// TwinCAT 3 PLC project PLC1
// Title: Project Title
// Company: Company Name
// ProjectVersion: 0.0.1.1
// ProgramVersion: 3.1.4024.0
// CompilerDefines: VISU_USEWSTRING
// libraries:
//   CmpBitmapPool, * (System)
//   FloatingPointUtils, * (System)
//   Tc2_EtherCAT, * (Beckhoff Automation GmbH)
//   Tc2_Math, * (Beckhoff Automation GmbH)
//   Tc2_MC2, * (Beckhoff Automation GmbH)
//   Tc2_Standard, * (Beckhoff Automation GmbH)
//   Tc2_System, * (Beckhoff Automation GmbH)
//   Tc2_Utilities, * (Beckhoff Automation GmbH)
//   Tc3_Module, * (Beckhoff Automation GmbH)
//   VisuDialogs, * (System)
//   Util,3.5.11.0,System
//   VisuSymbols,3.5.10.0,System
// project tree:
//   Data Collection/dataAnalyse/ E_BoxResultCode.TcDUT, E_WallEntryRule.TcDUT, FB_Window.TcPOU, prgDataAnaylse.TcPOU, ST_BoxCorner.TcDUT, ST_WallPermission.TcDUT
//   Data Collection/ dataGrab.TcGVL, Dat_550_DataAxis.TcVIS, prgDataGrab.TcPOU, structAnalysis.TcDUT, typeDataAxis.TcDUT, typeVectorOptions.TcDUT
//   Data Collection/dynamicBox/ diaDataBox.TcVIS, FB_BoxControl.TcPOU, structBoxData.TcDUT, textListLeft.TcTLO, textListRight.TcTLO, textListTop.TcTLO, textListBottom.TcTLO
//   Data Collection/task/ DataGrab_1.TcTTO, taskDataGrab.TcPOU, typePoints.TcDUT
//   HMI1/Data/ gLicenceView.TcGVL, gModeAlternate.TcGVL, ManualPageTitle.TcTLO, ModeRowText.TcTLO, ScreenNames.TcTLO, stationLinked.TcTLO, TaskText.TcTLO, CycleType.TcTLO, FaultState.TcTLO, flag.TcIPO (not stored), FlasherCorner.TcIPO (not stored), gHMIButtons.TcGVL, gHMIDataConst.TcGVL, gHMIMotionRows.TcGVL, gHMIUnits.TcGVL, gMsgView.TcGVL, HMIColour.TcGVL, HomeState.TcTLO, ModeStates.TcTLO, ModeStatesHeader.TcTLO, UnitRowText.TcTLO, MotionRowText.TcTLO, LanguageRowText.TcTLO, gHMIData.TcGVL, MotionRowImages.TcIPO (not stored)
//   HMI1/Data/TOAST-HMI/ gTOASTHMI.TcGVL, structHMI.TcDUT, structHMIBtns.TcDUT, structHMIGlobal.TcDUT, structHMIMessages.TcDUT
//   HMI1/Logic/ FB_ReadTextList.TcPOU, prgHMIaxis.TcPOU, prgModeRows.TcPOU, prgMotionRow.TcPOU, VisuInit.TcPOU, FB_FindTextIndexNum.TcPOU, FB_FindTextLangText.TcPOU, FC_Setup.TcPOU, pouHMI.TcPOU, prgHMIcontrol.TcPOU, prgHMIstations.TcPOU, prgHMIUnits.TcPOU, prgHMILanguage.TcPOU, prgReadTextList.TcPOU, prgShowButtons.TcPOU
//   HMI1/Screens/Diagnostic Fieldbus/EtherCAT/ diagEtherCATSlave.TcVIS (not stored), diagEtherCATSlaveDetail.TcVIS (not stored), Dia_801_EtherCAT.TcVIS (not stored)
//   HMI1/Screens/Diagnostic Fieldbus/PROFIBUS/ diagDPhelp.TcVIS (not stored), diagDPSlave.TcVIS (not stored), Dia_802_Profibus.TcVIS (not stored)
//   HMI1/Screens/Diagnostic Fieldbus/PROFINET/ diagProfiNetSlaveDetail.TcVIS (not stored), diagProfiNetSlave.TcVIS (not stored), Dia_803_ProfiNet.TcVIS (not stored)
//   HMI1/Screens/Diagnostic IO View/ Dia_800_DataDisplay.TcVIS
//   HMI1/Screens/Dialogs/ dialogEnterValueInteger.TcVIS, dialogReject.TcVIS, dialogDeviceInfo.TcVIS, dialogGetLicensesEx.TcVIS, dialogEnterValue.TcVIS, visuDataDisplay.TcVIS, visuTaskData.TcVIS, dialogStation.TcVIS
//   HMI1/Screens/Layout/ Lay_040_MachineLayout.TcVIS
//   HMI1/Screens/Machine Settings/ constCSV.TcGVL, FB_ReadParams.TcPOU, FB_WriteParams.TcPOU, MachineSettings.TcGVL, MaS_800_SettingScreen.TcVIS, pouMachineSettings.TcPOU, typeRecord.TcDUT, typeSettings.TcDUT
//   HMI1/Screens/Menu/ Men_030_MenuScreen.TcVIS, Men_031_MenuScreen_2.TcVIS, Men_032_MenuScreen_3.TcVIS
//   HMI1/Screens/Messages/ Msg_020_Alarms.TcVIS, Msg_021_AlarmsView.TcVIS
//   HMI1/Screens/Mode/ Mod_001_ModeScreen.TcVIS, Mod_101_ModeScreen_Alternate.TcVIS, Mod_002_ModeScreenRows.TcVIS
//   HMI1/Screens/Motion/ Mot_010_Motions.TcVIS, Mot_011_Axis.TcVIS
//   HMI1/Screens/Popup/ PopupMenu1.TcVIS, PopupMenu2.TcVIS, PopupMenu3.TcVIS, PopupMenu4.TcVIS, PopupMenu5.TcVIS, popup_test.TcVIS (not stored)
//   HMI1/Screens/Process/ Prc_500_Part.TcVIS (not stored), Prc_501_Cycle.TcVIS (not stored)
//   HMI1/Screens/Safety/ Saf_700_SafetyStatus.TcVIS (not stored), Saf_701_SafetyChecksum.TcVIS (not stored), visuSafetyRow.TcVIS (not stored)
//   HMI1/Screens/Sequences/ AutoRowsVisu.TcGVL, SeqTest.TcVIS (not stored)
//   HMI1/Screens/System/ Sys_900_About.TcVIS (not stored), Sys_902_Version.TcVIS (not stored), Sys_901_HMISystem.TcVIS (not stored)
//   HMI1/Screens/Units/ Unt_401_Units.TcVIS (not stored), Unt_402_Axis.TcVIS (not stored), Unt_403_Language.TcVIS (not stored)
//   HMI1/Screens/Web/ Web_300_Browser.TcVIS (not stored)
//   HMI1/Templates/ AxisRow.TcVIS, LanguageRow.TcVIS, ModeRow.TcVIS, Tmp_001_Template_Alternate.TcVIS, UnitRow.TcVIS, MotionRow.TcVIS, Tmp_000_Template.TcVIS, MessageRow.TcVIS
//   PLC/FBs/Diagnostic/EtherCAT/ enumEtherCATstate.TcGVL (not stored), enumEtherCATSuffix.TcGVL (not stored), etherCATdiag.TcGVL (not stored), ethercatImages.TcIPO (not stored), etherCATmasters.TcGVL (not stored), FB_CheckEC_CRC_errors.TcPOU (not stored), FB_DecodeEtherCAT.TcPOU (not stored), pouEtherCATDiag.TcPOU (not stored)
//   PLC/FBs/Diagnostic/Profibus/ pouDPDiag.TcPOU (not stored), profibusDiag.TcGVL (not stored), profibusImages.TcIPO (not stored)
//   PLC/FBs/Diagnostic/ProfiNet/ enumProfiNetState.TcGVL (not stored), enumProfiNetSuffix.TcGVL (not stored), FB_DecodePROFINET.TcPOU (not stored), pouPROFINETdiag.TcPOU (not stored), ProfiNetDiag.TcGVL (not stored), ProfiNETImages.TcIPO (not stored)
//   PLC/FBs/FBs/ FB_ApplyLocks.TcPOU (not stored), FB_CheckAnyMode.TcPOU (not stored), FB_Flasher.TcPOU, FB_HMI_Control_NoGroupRef.TcPOU (not stored), FB_PowerDelay.TcPOU (not stored), FB_StationStats.TcPOU (not stored), FB_Step.TcPOU (not stored), FB_CheckMessageBounds.TcPOU (not stored), FB_HMI_Control.TcPOU (not stored), FB_Mode.TcPOU (not stored), FB_PartBuild.TcPOU (not stored), FB_ModeStateToColour.TcPOU (not stored)
//   PLC/FBs/FCs/ FC_NOT.TcPOU (not stored)
//   PLC/FBs/IO View/ FB_DataCombine.TcPOU (not stored), ioView.TcGVL (not stored), pouDataDisplay.TcPOU (not stored), prgMemPointerView.TcPOU (not stored)
//   PLC/FBs/Robot/ FB_RobotComms.TcPOU (not stored), FB_RobotMotion.TcPOU (not stored), robotCall.TcPOU (not stored), robotGlobals.TcGVL (not stored), structRobot.TcDUT (not stored), structRobotInputs.TcDUT (not stored), structRobotOutputs.TcDUT (not stored)
//   PLC/FBs/Sequence/ typeAutoRowMotion.TcDUT (not stored), AutoRows.TcGVL (not stored), FB_GetStateAutoRow.TcPOU (not stored), typeRowHolder.TcDUT (not stored), typeSeqRow.TcDUT (not stored)
//   PLC/FBs/Tasks/ FB_CheckTasks.TcPOU (not stored), FB_Task.TcPOU (not stored), FC_S1_AssignTaskTimes.TcPOU (not stored), FC_S2_AssignTaskTimes.TcPOU (not stored), FC_S3_AssignTaskTimes.TcPOU (not stored), FC_S4_AssignTaskTimes.TcPOU (not stored), FC_S5_AssignTaskTimes.TcPOU (not stored), FC_S6_AssignTaskTimes.TcPOU (not stored)
//   PLC/Machine/Base/ Mc_Variant.TcGVL (not stored), Mc_Global.TcGVL (not stored), pouMachine.TcPOU (not stored)
//   PLC/Machine/Station 1/Motions/Screen 10/ S1_01_Motion_89.TcPOU (not stored), S1_01_Motion_90.TcPOU (not stored), S1_01_Motion_91.TcPOU (not stored), S1_01_Motion_92.TcPOU (not stored), S1_01_Motion_93.TcPOU (not stored), S1_01_Motion_94.TcPOU (not stored), S1_01_Motion_95.TcPOU (not stored), S1_01_Motion_96.TcPOU (not stored), S1_01_Motion_97.TcPOU (not stored), S1_01_Motion_98.TcPOU (not stored), S1_01_Motion_99.TcPOU (not stored)
//   PLC/Machine/Station 1/Motions/Screen 1/ S1_01_RobPickPart_1.TcPOU (not stored), S1_01_RobClamp1_2.TcPOU (not stored), S1_01_RobClamp2_3.TcPOU (not stored), S1_01_RobWash_4.TcPOU (not stored), S1_01_WasherJets_5.TcPOU (not stored), S1_01_RobMarker_6.TcPOU (not stored), S1_01_MarkPart_7.TcPOU (not stored), S1_01_Motion_8.TcPOU (not stored), S1_01_Motion_9.TcPOU (not stored)
//   PLC/Machine/Station 1/Motions/Screen 2/ S1_01_Motion_10.TcPOU (not stored), S1_01_Motion_11.TcPOU (not stored), S1_01_Motion_12.TcPOU (not stored), S1_01_Motion_13.TcPOU (not stored), S1_01_Motion_14.TcPOU (not stored), S1_01_Motion_15.TcPOU (not stored), S1_01_Motion_16.TcPOU (not stored), S1_01_Motion_17.TcPOU (not stored), S1_01_Motion_18.TcPOU (not stored), S1_01_Motion_19.TcPOU (not stored)
//   PLC/Machine/Station 1/Motions/Screen 3/ S1_01_Motion_20.TcPOU (not stored), S1_01_Motion_21.TcPOU (not stored), S1_01_Motion_22.TcPOU (not stored), S1_01_Motion_23.TcPOU (not stored), S1_01_Motion_24.TcPOU (not stored), S1_01_Motion_25.TcPOU (not stored), S1_01_Motion_26.TcPOU (not stored), S1_01_Motion_27.TcPOU (not stored), S1_01_Motion_28.TcPOU (not stored)
//   PLC/Machine/Station 1/Motions/Screen 4/ S1_01_Motion_29.TcPOU (not stored), S1_01_Motion_30.TcPOU (not stored), S1_01_Motion_31.TcPOU (not stored), S1_01_Motion_32.TcPOU (not stored), S1_01_Motion_33.TcPOU (not stored), S1_01_Motion_34.TcPOU (not stored), S1_01_Motion_35.TcPOU (not stored), S1_01_Motion_36.TcPOU (not stored), S1_01_Motion_37.TcPOU (not stored), S1_01_Motion_38.TcPOU (not stored)
//   PLC/Machine/Station 1/Motions/Screen 5/ S1_01_Motion_39.TcPOU (not stored), S1_01_Motion_40.TcPOU (not stored), S1_01_Motion_41.TcPOU (not stored), S1_01_Motion_42.TcPOU (not stored), S1_01_Motion_43.TcPOU (not stored), S1_01_Motion_44.TcPOU (not stored), S1_01_Motion_45.TcPOU (not stored), S1_01_Motion_46.TcPOU (not stored), S1_01_Motion_47.TcPOU (not stored), S1_01_Motion_48.TcPOU (not stored)
//   PLC/Machine/Station 1/Motions/Screen 6/ S1_01_Motion_49.TcPOU (not stored), S1_01_Motion_50.TcPOU (not stored), S1_01_Motion_51.TcPOU (not stored), S1_01_Motion_52.TcPOU (not stored), S1_01_Motion_53.TcPOU (not stored), S1_01_Motion_54.TcPOU (not stored), S1_01_Motion_55.TcPOU (not stored), S1_01_Motion_56.TcPOU (not stored), S1_01_Motion_57.TcPOU (not stored), S1_01_Motion_58.TcPOU (not stored)
//   PLC/Machine/Station 1/Motions/Screen 7/ S1_01_Motion_59.TcPOU (not stored), S1_01_Motion_60.TcPOU (not stored), S1_01_Motion_61.TcPOU (not stored), S1_01_Motion_62.TcPOU (not stored), S1_01_Motion_63.TcPOU (not stored), S1_01_Motion_64.TcPOU (not stored), S1_01_Motion_65.TcPOU (not stored), S1_01_Motion_66.TcPOU (not stored), S1_01_Motion_67.TcPOU (not stored), S1_01_Motion_68.TcPOU (not stored)
//   PLC/Machine/Station 1/Motions/Screen 8/ S1_01_Motion_69.TcPOU (not stored), S1_01_Motion_70.TcPOU (not stored), S1_01_Motion_71.TcPOU (not stored), S1_01_Motion_72.TcPOU (not stored), S1_01_Motion_73.TcPOU (not stored), S1_01_Motion_74.TcPOU (not stored), S1_01_Motion_75.TcPOU (not stored), S1_01_Motion_76.TcPOU (not stored), S1_01_Motion_77.TcPOU (not stored), S1_01_Motion_78.TcPOU (not stored)
//   PLC/Machine/Station 1/Motions/Screen 9/ S1_01_Motion_79.TcPOU (not stored), S1_01_Motion_80.TcPOU (not stored), S1_01_Motion_81.TcPOU (not stored), S1_01_Motion_82.TcPOU (not stored), S1_01_Motion_83.TcPOU (not stored), S1_01_Motion_84.TcPOU (not stored), S1_01_Motion_85.TcPOU (not stored), S1_01_Motion_86.TcPOU (not stored), S1_01_Motion_87.TcPOU (not stored), S1_01_Motion_88.TcPOU (not stored)
//   PLC/Machine/Station 1/Sequence/ FB_S1_Sequence.TcPOU (not stored), S1sfc.TcGVL (not stored), struct_SFC_Row.TcDUT (not stored)
//   PLC/Machine/Station 2/Motions/Screen 10/ S2_01_Motion_89.TcPOU (not stored), S2_01_Motion_90.TcPOU (not stored), S2_01_Motion_91.TcPOU (not stored), S2_01_Motion_92.TcPOU (not stored), S2_01_Motion_93.TcPOU (not stored), S2_01_Motion_94.TcPOU (not stored), S2_01_Motion_95.TcPOU (not stored), S2_01_Motion_96.TcPOU (not stored), S2_01_Motion_97.TcPOU (not stored), S2_01_Motion_98.TcPOU (not stored), S2_01_Motion_99.TcPOU (not stored)
//   PLC/Machine/Station 2/Motions/Screen 1/ S2_01_Motion_1.TcPOU (not stored), S2_01_Motion_2.TcPOU (not stored), S2_01_Motion_3.TcPOU (not stored), S2_01_Motion_4.TcPOU (not stored), S2_01_Motion_5.TcPOU (not stored), S2_01_Motion_6.TcPOU (not stored), S2_01_Motion_7.TcPOU (not stored), S2_01_Motion_8.TcPOU (not stored), S2_01_Motion_9.TcPOU (not stored)
//   PLC/Machine/Station 2/Motions/Screen 2/ S2_01_Motion_10.TcPOU (not stored), S2_01_Motion_11.TcPOU (not stored), S2_01_Motion_12.TcPOU (not stored), S2_01_Motion_13.TcPOU (not stored), S2_01_Motion_14.TcPOU (not stored), S2_01_Motion_15.TcPOU (not stored), S2_01_Motion_16.TcPOU (not stored), S2_01_Motion_17.TcPOU (not stored), S2_01_Motion_18.TcPOU (not stored), S2_01_Motion_19.TcPOU (not stored)
//   PLC/Machine/Station 2/Motions/Screen 3/ S2_01_Motion_20.TcPOU (not stored), S2_01_Motion_21.TcPOU (not stored), S2_01_Motion_22.TcPOU (not stored), S2_01_Motion_23.TcPOU (not stored), S2_01_Motion_24.TcPOU (not stored), S2_01_Motion_25.TcPOU (not stored), S2_01_Motion_26.TcPOU (not stored), S2_01_Motion_27.TcPOU (not stored), S2_01_Motion_28.TcPOU (not stored)
//   PLC/Machine/Station 2/Motions/Screen 4/ S2_01_Motion_29.TcPOU (not stored), S2_01_Motion_30.TcPOU (not stored), S2_01_Motion_31.TcPOU (not stored), S2_01_Motion_32.TcPOU (not stored), S2_01_Motion_33.TcPOU (not stored), S2_01_Motion_34.TcPOU (not stored), S2_01_Motion_35.TcPOU (not stored), S2_01_Motion_36.TcPOU (not stored), S2_01_Motion_37.TcPOU (not stored), S2_01_Motion_38.TcPOU (not stored)
//   PLC/Machine/Station 2/Motions/Screen 5/ S2_01_Motion_39.TcPOU (not stored), S2_01_Motion_40.TcPOU (not stored), S2_01_Motion_41.TcPOU (not stored), S2_01_Motion_42.TcPOU (not stored), S2_01_Motion_43.TcPOU (not stored), S2_01_Motion_44.TcPOU (not stored), S2_01_Motion_45.TcPOU (not stored), S2_01_Motion_46.TcPOU (not stored), S2_01_Motion_47.TcPOU (not stored), S2_01_Motion_48.TcPOU (not stored)
//   PLC/Machine/Station 2/Motions/Screen 6/ S2_01_Motion_49.TcPOU (not stored), S2_01_Motion_50.TcPOU (not stored), S2_01_Motion_51.TcPOU (not stored), S2_01_Motion_52.TcPOU (not stored), S2_01_Motion_53.TcPOU (not stored), S2_01_Motion_54.TcPOU (not stored), S2_01_Motion_55.TcPOU (not stored), S2_01_Motion_56.TcPOU (not stored), S2_01_Motion_57.TcPOU (not stored), S2_01_Motion_58.TcPOU (not stored)
//   PLC/Machine/Station 2/Motions/Screen 7/ S2_01_Motion_59.TcPOU (not stored), S2_01_Motion_60.TcPOU (not stored), S2_01_Motion_61.TcPOU (not stored), S2_01_Motion_62.TcPOU (not stored), S2_01_Motion_63.TcPOU (not stored), S2_01_Motion_64.TcPOU (not stored), S2_01_Motion_65.TcPOU (not stored), S2_01_Motion_66.TcPOU (not stored), S2_01_Motion_67.TcPOU (not stored), S2_01_Motion_68.TcPOU (not stored)
//   PLC/Machine/Station 2/Motions/Screen 8/ S2_01_Motion_69.TcPOU (not stored), S2_01_Motion_70.TcPOU (not stored), S2_01_Motion_71.TcPOU (not stored), S2_01_Motion_72.TcPOU (not stored), S2_01_Motion_73.TcPOU (not stored), S2_01_Motion_74.TcPOU (not stored), S2_01_Motion_75.TcPOU (not stored), S2_01_Motion_76.TcPOU (not stored), S2_01_Motion_77.TcPOU (not stored), S2_01_Motion_78.TcPOU (not stored)
//   PLC/Machine/Station 2/Motions/Screen 9/ S2_01_Motion_79.TcPOU (not stored), S2_01_Motion_80.TcPOU (not stored), S2_01_Motion_81.TcPOU (not stored), S2_01_Motion_82.TcPOU (not stored), S2_01_Motion_83.TcPOU (not stored), S2_01_Motion_84.TcPOU (not stored), S2_01_Motion_85.TcPOU (not stored), S2_01_Motion_86.TcPOU (not stored), S2_01_Motion_87.TcPOU (not stored), S2_01_Motion_88.TcPOU (not stored)
//   PLC/Machine/Station 3/Motions/Screen 10/ S3_01_Motion_89.TcPOU (not stored), S3_01_Motion_90.TcPOU (not stored), S3_01_Motion_91.TcPOU (not stored), S3_01_Motion_92.TcPOU (not stored), S3_01_Motion_93.TcPOU (not stored), S3_01_Motion_94.TcPOU (not stored), S3_01_Motion_95.TcPOU (not stored), S3_01_Motion_96.TcPOU (not stored), S3_01_Motion_97.TcPOU (not stored), S3_01_Motion_98.TcPOU (not stored), S3_01_Motion_99.TcPOU (not stored)
//   PLC/Machine/Station 3/Motions/Screen 1/ S3_01_Motion_1.TcPOU (not stored), S3_01_Motion_2.TcPOU (not stored), S3_01_Motion_3.TcPOU (not stored), S3_01_Motion_4.TcPOU (not stored), S3_01_Motion_5.TcPOU (not stored), S3_01_Motion_6.TcPOU (not stored), S3_01_Motion_7.TcPOU (not stored), S3_01_Motion_8.TcPOU (not stored), S3_01_Motion_9.TcPOU (not stored)
//   PLC/Machine/Station 3/Motions/Screen 2/ S3_01_Motion_10.TcPOU (not stored), S3_01_Motion_11.TcPOU (not stored), S3_01_Motion_12.TcPOU (not stored), S3_01_Motion_13.TcPOU (not stored), S3_01_Motion_14.TcPOU (not stored), S3_01_Motion_15.TcPOU (not stored), S3_01_Motion_16.TcPOU (not stored), S3_01_Motion_17.TcPOU (not stored), S3_01_Motion_18.TcPOU (not stored), S3_01_Motion_19.TcPOU (not stored)
//   PLC/Machine/Station 3/Motions/Screen 3/ S3_01_Motion_20.TcPOU (not stored), S3_01_Motion_21.TcPOU (not stored), S3_01_Motion_22.TcPOU (not stored), S3_01_Motion_23.TcPOU (not stored), S3_01_Motion_24.TcPOU (not stored), S3_01_Motion_25.TcPOU (not stored), S3_01_Motion_26.TcPOU (not stored), S3_01_Motion_27.TcPOU (not stored), S3_01_Motion_28.TcPOU (not stored)
//   PLC/Machine/Station 3/Motions/Screen 4/ S3_01_Motion_29.TcPOU (not stored), S3_01_Motion_30.TcPOU (not stored), S3_01_Motion_31.TcPOU (not stored), S3_01_Motion_32.TcPOU (not stored), S3_01_Motion_33.TcPOU (not stored), S3_01_Motion_34.TcPOU (not stored), S3_01_Motion_35.TcPOU (not stored), S3_01_Motion_36.TcPOU (not stored), S3_01_Motion_37.TcPOU (not stored), S3_01_Motion_38.TcPOU (not stored)
//   PLC/Machine/Station 3/Motions/Screen 5/ S3_01_Motion_39.TcPOU (not stored), S3_01_Motion_40.TcPOU (not stored), S3_01_Motion_41.TcPOU (not stored), S3_01_Motion_42.TcPOU (not stored), S3_01_Motion_43.TcPOU (not stored), S3_01_Motion_44.TcPOU (not stored), S3_01_Motion_45.TcPOU (not stored), S3_01_Motion_46.TcPOU (not stored), S3_01_Motion_47.TcPOU (not stored), S3_01_Motion_48.TcPOU (not stored)
//   PLC/Machine/Station 3/Motions/Screen 6/ S3_01_Motion_49.TcPOU (not stored), S3_01_Motion_50.TcPOU (not stored), S3_01_Motion_51.TcPOU (not stored), S3_01_Motion_52.TcPOU (not stored), S3_01_Motion_53.TcPOU (not stored), S3_01_Motion_54.TcPOU (not stored), S3_01_Motion_55.TcPOU (not stored), S3_01_Motion_56.TcPOU (not stored), S3_01_Motion_57.TcPOU (not stored), S3_01_Motion_58.TcPOU (not stored)
//   PLC/Machine/Station 3/Motions/Screen 7/ S3_01_Motion_59.TcPOU (not stored), S3_01_Motion_60.TcPOU (not stored), S3_01_Motion_61.TcPOU (not stored), S3_01_Motion_62.TcPOU (not stored), S3_01_Motion_63.TcPOU (not stored), S3_01_Motion_64.TcPOU (not stored), S3_01_Motion_65.TcPOU (not stored), S3_01_Motion_66.TcPOU (not stored), S3_01_Motion_67.TcPOU (not stored), S3_01_Motion_68.TcPOU (not stored)
//   PLC/Machine/Station 3/Motions/Screen 8/ S3_01_Motion_69.TcPOU (not stored), S3_01_Motion_70.TcPOU (not stored), S3_01_Motion_71.TcPOU (not stored), S3_01_Motion_72.TcPOU (not stored), S3_01_Motion_73.TcPOU (not stored), S3_01_Motion_74.TcPOU (not stored), S3_01_Motion_75.TcPOU (not stored), S3_01_Motion_76.TcPOU (not stored), S3_01_Motion_77.TcPOU (not stored), S3_01_Motion_78.TcPOU (not stored)
//   PLC/Machine/Station 3/Motions/Screen 9/ S3_01_Motion_79.TcPOU (not stored), S3_01_Motion_80.TcPOU (not stored), S3_01_Motion_81.TcPOU (not stored), S3_01_Motion_82.TcPOU (not stored), S3_01_Motion_83.TcPOU (not stored), S3_01_Motion_84.TcPOU (not stored), S3_01_Motion_85.TcPOU (not stored), S3_01_Motion_86.TcPOU (not stored), S3_01_Motion_87.TcPOU (not stored), S3_01_Motion_88.TcPOU (not stored)
//   PLC/Machine/Station 4/Motions/Screen 10/ S4_01_Motion_89.TcPOU (not stored), S4_01_Motion_90.TcPOU (not stored), S4_01_Motion_91.TcPOU (not stored), S4_01_Motion_92.TcPOU (not stored), S4_01_Motion_93.TcPOU (not stored), S4_01_Motion_94.TcPOU (not stored), S4_01_Motion_95.TcPOU (not stored), S4_01_Motion_96.TcPOU (not stored), S4_01_Motion_97.TcPOU (not stored), S4_01_Motion_98.TcPOU (not stored), S4_01_Motion_99.TcPOU (not stored)
//   PLC/Machine/Station 4/Motions/Screen 1/ S4_01_Motion_1.TcPOU (not stored), S4_01_Motion_2.TcPOU (not stored), S4_01_Motion_3.TcPOU (not stored), S4_01_Motion_4.TcPOU (not stored), S4_01_Motion_5.TcPOU (not stored), S4_01_Motion_6.TcPOU (not stored), S4_01_Motion_7.TcPOU (not stored), S4_01_Motion_8.TcPOU (not stored), S4_01_Motion_9.TcPOU (not stored)
//   PLC/Machine/Station 4/Motions/Screen 2/ S4_01_Motion_10.TcPOU (not stored), S4_01_Motion_11.TcPOU (not stored), S4_01_Motion_12.TcPOU (not stored), S4_01_Motion_13.TcPOU (not stored), S4_01_Motion_14.TcPOU (not stored), S4_01_Motion_15.TcPOU (not stored), S4_01_Motion_16.TcPOU (not stored), S4_01_Motion_17.TcPOU (not stored), S4_01_Motion_18.TcPOU (not stored), S4_01_Motion_19.TcPOU (not stored)
//   PLC/Machine/Station 4/Motions/Screen 3/ S4_01_Motion_20.TcPOU (not stored), S4_01_Motion_21.TcPOU (not stored), S4_01_Motion_22.TcPOU (not stored), S4_01_Motion_23.TcPOU (not stored), S4_01_Motion_24.TcPOU (not stored), S4_01_Motion_25.TcPOU (not stored), S4_01_Motion_26.TcPOU (not stored), S4_01_Motion_27.TcPOU (not stored), S4_01_Motion_28.TcPOU (not stored)
//   PLC/Machine/Station 4/Motions/Screen 4/ S4_01_Motion_29.TcPOU (not stored), S4_01_Motion_30.TcPOU (not stored), S4_01_Motion_31.TcPOU (not stored), S4_01_Motion_32.TcPOU (not stored), S4_01_Motion_33.TcPOU (not stored), S4_01_Motion_34.TcPOU (not stored), S4_01_Motion_35.TcPOU (not stored), S4_01_Motion_36.TcPOU (not stored), S4_01_Motion_37.TcPOU (not stored), S4_01_Motion_38.TcPOU (not stored)
//   PLC/Machine/Station 4/Motions/Screen 5/ S4_01_Motion_39.TcPOU (not stored), S4_01_Motion_40.TcPOU (not stored), S4_01_Motion_41.TcPOU (not stored), S4_01_Motion_42.TcPOU (not stored), S4_01_Motion_43.TcPOU (not stored), S4_01_Motion_44.TcPOU (not stored), S4_01_Motion_45.TcPOU (not stored), S4_01_Motion_46.TcPOU (not stored), S4_01_Motion_47.TcPOU (not stored), S4_01_Motion_48.TcPOU (not stored)
//   PLC/Machine/Station 4/Motions/Screen 6/ S4_01_Motion_49.TcPOU (not stored), S4_01_Motion_50.TcPOU (not stored), S4_01_Motion_51.TcPOU (not stored), S4_01_Motion_52.TcPOU (not stored), S4_01_Motion_53.TcPOU (not stored), S4_01_Motion_54.TcPOU (not stored), S4_01_Motion_55.TcPOU (not stored), S4_01_Motion_56.TcPOU (not stored), S4_01_Motion_57.TcPOU (not stored), S4_01_Motion_58.TcPOU (not stored)
//   PLC/Machine/Station 4/Motions/Screen 7/ S4_01_Motion_59.TcPOU (not stored), S4_01_Motion_60.TcPOU (not stored), S4_01_Motion_61.TcPOU (not stored), S4_01_Motion_62.TcPOU (not stored), S4_01_Motion_63.TcPOU (not stored), S4_01_Motion_64.TcPOU (not stored), S4_01_Motion_65.TcPOU (not stored), S4_01_Motion_66.TcPOU (not stored), S4_01_Motion_67.TcPOU (not stored), S4_01_Motion_68.TcPOU (not stored)
//   PLC/Machine/Station 4/Motions/Screen 8/ S4_01_Motion_69.TcPOU (not stored), S4_01_Motion_70.TcPOU (not stored), S4_01_Motion_71.TcPOU (not stored), S4_01_Motion_72.TcPOU (not stored), S4_01_Motion_73.TcPOU (not stored), S4_01_Motion_74.TcPOU (not stored), S4_01_Motion_75.TcPOU (not stored), S4_01_Motion_76.TcPOU (not stored), S4_01_Motion_77.TcPOU (not stored), S4_01_Motion_78.TcPOU (not stored)
//   PLC/Machine/Station 4/Motions/Screen 9/ S4_01_Motion_79.TcPOU (not stored), S4_01_Motion_80.TcPOU (not stored), S4_01_Motion_81.TcPOU (not stored), S4_01_Motion_82.TcPOU (not stored), S4_01_Motion_83.TcPOU (not stored), S4_01_Motion_84.TcPOU (not stored), S4_01_Motion_85.TcPOU (not stored), S4_01_Motion_86.TcPOU (not stored), S4_01_Motion_87.TcPOU (not stored), S4_01_Motion_88.TcPOU (not stored)
//   PLC/Machine/Station 5/Motions/Screen 10/ S5_01_Motion_89.TcPOU (not stored), S5_01_Motion_90.TcPOU (not stored), S5_01_Motion_91.TcPOU (not stored), S5_01_Motion_92.TcPOU (not stored), S5_01_Motion_93.TcPOU (not stored), S5_01_Motion_94.TcPOU (not stored), S5_01_Motion_95.TcPOU (not stored), S5_01_Motion_96.TcPOU (not stored), S5_01_Motion_97.TcPOU (not stored), S5_01_Motion_98.TcPOU (not stored), S5_01_Motion_99.TcPOU (not stored)
//   PLC/Machine/Station 5/Motions/Screen 1/ S5_01_Motion_1.TcPOU (not stored), S5_01_Motion_2.TcPOU (not stored), S5_01_Motion_3.TcPOU (not stored), S5_01_Motion_4.TcPOU (not stored), S5_01_Motion_5.TcPOU (not stored), S5_01_Motion_6.TcPOU (not stored), S5_01_Motion_7.TcPOU (not stored), S5_01_Motion_8.TcPOU (not stored), S5_01_Motion_9.TcPOU (not stored)
//   PLC/Machine/Station 5/Motions/Screen 2/ S5_01_Motion_10.TcPOU (not stored), S5_01_Motion_11.TcPOU (not stored), S5_01_Motion_12.TcPOU (not stored), S5_01_Motion_13.TcPOU (not stored), S5_01_Motion_14.TcPOU (not stored), S5_01_Motion_15.TcPOU (not stored), S5_01_Motion_16.TcPOU (not stored), S5_01_Motion_17.TcPOU (not stored), S5_01_Motion_18.TcPOU (not stored), S5_01_Motion_19.TcPOU (not stored)
//   PLC/Machine/Station 5/Motions/Screen 3/ S5_01_Motion_20.TcPOU (not stored), S5_01_Motion_21.TcPOU (not stored), S5_01_Motion_22.TcPOU (not stored), S5_01_Motion_23.TcPOU (not stored), S5_01_Motion_24.TcPOU (not stored), S5_01_Motion_25.TcPOU (not stored), S5_01_Motion_26.TcPOU (not stored), S5_01_Motion_27.TcPOU (not stored), S5_01_Motion_28.TcPOU (not stored), S5_01_Motion_29.TcPOU (not stored)
//   PLC/Machine/Station 5/Motions/Screen 4/ S5_01_Motion_30.TcPOU (not stored), S5_01_Motion_31.TcPOU (not stored), S5_01_Motion_32.TcPOU (not stored), S5_01_Motion_33.TcPOU (not stored), S5_01_Motion_34.TcPOU (not stored), S5_01_Motion_35.TcPOU (not stored), S5_01_Motion_36.TcPOU (not stored), S5_01_Motion_37.TcPOU (not stored), S5_01_Motion_38.TcPOU (not stored), S5_01_Motion_39.TcPOU (not stored)
//   PLC/Machine/Station 5/Motions/Screen 5/ S5_01_Motion_40.TcPOU (not stored), S5_01_Motion_41.TcPOU (not stored), S5_01_Motion_42.TcPOU (not stored), S5_01_Motion_43.TcPOU (not stored), S5_01_Motion_44.TcPOU (not stored), S5_01_Motion_45.TcPOU (not stored), S5_01_Motion_46.TcPOU (not stored), S5_01_Motion_47.TcPOU (not stored), S5_01_Motion_48.TcPOU (not stored), S5_01_Motion_49.TcPOU (not stored)
//   PLC/Machine/Station 5/Motions/Screen 6/ S5_01_Motion_50.TcPOU (not stored), S5_01_Motion_51.TcPOU (not stored), S5_01_Motion_52.TcPOU (not stored), S5_01_Motion_53.TcPOU (not stored), S5_01_Motion_54.TcPOU (not stored), S5_01_Motion_55.TcPOU (not stored), S5_01_Motion_56.TcPOU (not stored), S5_01_Motion_57.TcPOU (not stored), S5_01_Motion_58.TcPOU (not stored), S5_01_Motion_59.TcPOU (not stored)
//   PLC/Machine/Station 5/Motions/Screen 7/ S5_01_Motion_60.TcPOU (not stored), S5_01_Motion_61.TcPOU (not stored), S5_01_Motion_62.TcPOU (not stored), S5_01_Motion_63.TcPOU (not stored), S5_01_Motion_64.TcPOU (not stored), S5_01_Motion_65.TcPOU (not stored), S5_01_Motion_66.TcPOU (not stored), S5_01_Motion_67.TcPOU (not stored), S5_01_Motion_68.TcPOU (not stored), S5_01_Motion_69.TcPOU (not stored)
//   PLC/Machine/Station 5/Motions/Screen 8/ S5_01_Motion_70.TcPOU (not stored), S5_01_Motion_71.TcPOU (not stored), S5_01_Motion_72.TcPOU (not stored), S5_01_Motion_73.TcPOU (not stored), S5_01_Motion_74.TcPOU (not stored), S5_01_Motion_75.TcPOU (not stored), S5_01_Motion_76.TcPOU (not stored), S5_01_Motion_77.TcPOU (not stored), S5_01_Motion_78.TcPOU (not stored), S5_01_Motion_79.TcPOU (not stored)
//   PLC/Machine/Station 5/Motions/Screen 9/ S5_01_Motion_80.TcPOU (not stored), S5_01_Motion_81.TcPOU (not stored), S5_01_Motion_82.TcPOU (not stored), S5_01_Motion_83.TcPOU (not stored), S5_01_Motion_84.TcPOU (not stored), S5_01_Motion_85.TcPOU (not stored), S5_01_Motion_86.TcPOU (not stored), S5_01_Motion_87.TcPOU (not stored), S5_01_Motion_88.TcPOU (not stored)
//   PLC/Machine/Station 6/Motions/Screen 10/ S6_01_Motion_89.TcPOU (not stored), S6_01_Motion_90.TcPOU (not stored), S6_01_Motion_91.TcPOU (not stored), S6_01_Motion_92.TcPOU (not stored), S6_01_Motion_93.TcPOU (not stored), S6_01_Motion_94.TcPOU (not stored), S6_01_Motion_95.TcPOU (not stored), S6_01_Motion_96.TcPOU (not stored), S6_01_Motion_97.TcPOU (not stored), S6_01_Motion_98.TcPOU (not stored), S6_01_Motion_99.TcPOU (not stored)
//   PLC/Machine/Station 6/Motions/Screen 1/ S6_01_Motion_1.TcPOU (not stored), S6_01_Motion_2.TcPOU (not stored), S6_01_Motion_3.TcPOU (not stored), S6_01_Motion_4.TcPOU (not stored), S6_01_Motion_5.TcPOU (not stored), S6_01_Motion_6.TcPOU (not stored), S6_01_Motion_7.TcPOU (not stored), S6_01_Motion_8.TcPOU (not stored), S6_01_Motion_9.TcPOU (not stored)
//   PLC/Machine/Station 6/Motions/Screen 2/ S6_01_Motion_10.TcPOU (not stored), S6_01_Motion_11.TcPOU (not stored), S6_01_Motion_12.TcPOU (not stored), S6_01_Motion_13.TcPOU (not stored), S6_01_Motion_14.TcPOU (not stored), S6_01_Motion_15.TcPOU (not stored), S6_01_Motion_16.TcPOU (not stored), S6_01_Motion_17.TcPOU (not stored), S6_01_Motion_18.TcPOU (not stored), S6_01_Motion_19.TcPOU (not stored)
//   PLC/Machine/Station 6/Motions/Screen 3/ S6_01_Motion_20.TcPOU (not stored), S6_01_Motion_21.TcPOU (not stored), S6_01_Motion_22.TcPOU (not stored), S6_01_Motion_23.TcPOU (not stored), S6_01_Motion_24.TcPOU (not stored), S6_01_Motion_25.TcPOU (not stored), S6_01_Motion_26.TcPOU (not stored), S6_01_Motion_27.TcPOU (not stored), S6_01_Motion_28.TcPOU (not stored), S6_01_Motion_29.TcPOU (not stored)
//   PLC/Machine/Station 6/Motions/Screen 4/ S6_01_Motion_30.TcPOU (not stored), S6_01_Motion_31.TcPOU (not stored), S6_01_Motion_32.TcPOU (not stored), S6_01_Motion_33.TcPOU (not stored), S6_01_Motion_34.TcPOU (not stored), S6_01_Motion_35.TcPOU (not stored), S6_01_Motion_36.TcPOU (not stored), S6_01_Motion_37.TcPOU (not stored), S6_01_Motion_38.TcPOU (not stored), S6_01_Motion_39.TcPOU (not stored)
//   PLC/Machine/Station 6/Motions/Screen 5/ S6_01_Motion_40.TcPOU (not stored), S6_01_Motion_41.TcPOU (not stored), S6_01_Motion_42.TcPOU (not stored), S6_01_Motion_43.TcPOU (not stored), S6_01_Motion_44.TcPOU (not stored), S6_01_Motion_45.TcPOU (not stored), S6_01_Motion_46.TcPOU (not stored), S6_01_Motion_47.TcPOU (not stored), S6_01_Motion_48.TcPOU (not stored), S6_01_Motion_49.TcPOU (not stored)
//   PLC/Machine/Station 6/Motions/Screen 6/ S6_01_Motion_50.TcPOU (not stored), S6_01_Motion_51.TcPOU (not stored), S6_01_Motion_52.TcPOU (not stored), S6_01_Motion_53.TcPOU (not stored), S6_01_Motion_54.TcPOU (not stored), S6_01_Motion_55.TcPOU (not stored), S6_01_Motion_56.TcPOU (not stored), S6_01_Motion_57.TcPOU (not stored), S6_01_Motion_58.TcPOU (not stored), S6_01_Motion_59.TcPOU (not stored)
//   PLC/Machine/Station 6/Motions/Screen 7/ S6_01_Motion_60.TcPOU (not stored), S6_01_Motion_61.TcPOU (not stored), S6_01_Motion_62.TcPOU (not stored), S6_01_Motion_63.TcPOU (not stored), S6_01_Motion_64.TcPOU (not stored), S6_01_Motion_65.TcPOU (not stored), S6_01_Motion_66.TcPOU (not stored), S6_01_Motion_67.TcPOU (not stored), S6_01_Motion_68.TcPOU (not stored), S6_01_Motion_69.TcPOU (not stored)
//   PLC/Machine/Station 6/Motions/Screen 8/ S6_01_Motion_70.TcPOU (not stored), S6_01_Motion_71.TcPOU (not stored), S6_01_Motion_72.TcPOU (not stored), S6_01_Motion_73.TcPOU (not stored), S6_01_Motion_74.TcPOU (not stored), S6_01_Motion_75.TcPOU (not stored), S6_01_Motion_76.TcPOU (not stored), S6_01_Motion_77.TcPOU (not stored), S6_01_Motion_78.TcPOU (not stored), S6_01_Motion_79.TcPOU (not stored)
//   PLC/Machine/Station 6/Motions/Screen 9/ S6_01_Motion_80.TcPOU (not stored), S6_01_Motion_81.TcPOU (not stored), S6_01_Motion_82.TcPOU (not stored), S6_01_Motion_83.TcPOU (not stored), S6_01_Motion_84.TcPOU (not stored), S6_01_Motion_85.TcPOU (not stored), S6_01_Motion_86.TcPOU (not stored), S6_01_Motion_87.TcPOU (not stored), S6_01_Motion_88.TcPOU (not stored)
//   PLC/Safety/ enumEstopState.TcDUT, prgSafetyMain.TcPOU, Safety.TcGVL, structEstopDiag.TcDUT, structSafetyEstopDiagBOOList.TcDUT
//   PLC/System/ImplicitChecks/ CheckBounds.TcPOU (not stored), CheckDivDInt.TcPOU (not stored), CheckDivLInt.TcPOU (not stored), CheckDivLReal.TcPOU (not stored), CheckDivReal.TcPOU (not stored), CheckLRangeSigned.TcPOU (not stored), CheckLRangeUnsigned.TcPOU (not stored), CheckPointer.TcPOU (not stored), CheckRangeSigned.TcPOU (not stored), CheckRangeUnsigned.TcPOU (not stored)
//   Project Information/ F_GetCompany.TcPOU, F_GetTitle.TcPOU, F_GetVersion.TcPOU
//   Version/ Global_Version.TcGVL
//   X_DUTs/Diagnostic/ typeDPSlaveIndicator.TcDUT, typeEtherCATIndicator.TcDUT, typeEtherCATmasters.TcDUT, typeEtherCATState.TcDUT, typePROFINETIndicator.TcDUT, typeProfiNetMaster.TcDUT, typePROFINETState.TcDUT
//   X_DUTs/Drives/ HMIaxisDefinition.TcDUT, typeDriveInterface.TcDUT
//   X_DUTs/HMI/ typeBtnFdbk.TcDUT, typeBtnHides.TcDUT, typeBtnPress.TcDUT, typeHMIheader.TcDUT, typeMessageRow.TcDUT (not stored), typeMessageRowsArry.TcDUT, typeStationEnables.TcDUT (not stored)
//   X_DUTs/IO View/ dutDWord.TcDUT (not stored), typeCombineString.TcDUT (not stored)
//   X_DUTs/Langauge/ LanguageLocation.TcDUT (not stored)
//   X_DUTs/MessageView/ typeNewMsg.TcDUT, typeNewMsgHeader.TcDUT (not stored), typeNewMsgStyle.TcDUT
//   X_DUTs/Message/ typeAlarmViewStation.TcDUT (not stored), typeMessage.TcDUT (not stored), typeStationMessage.TcDUT (not stored), typeStationStatus.TcDUT (not stored)
//   X_DUTs/Motion/ RowConfig.TcDUT (not stored), typeMotionRecordRow.TcDUT, typeMotionRow.TcDUT, typeMotionRowArry.TcDUT, typeMotionRowButtons.TcDUT, typeMotionRowIO.TcDUT, typeMotionSide.TcDUT
//   X_DUTs/Screen/ typeMotionScreen.TcDUT, typeMotionScreenBtn.TcDUT
//   X_DUTs/Setup/ typeSetupMachine.TcDUT (not stored), typeSetupStation.TcDUT
//   X_DUTs/Station/ enumStationState.TcDUT, typeIndividualTask.TcDUT, typeRemote.TcDUT (not stored), typeStation.TcDUT, typeStationComplexity.TcDUT, typeStationComplexityBuffer.TcDUT, typeStationLockModes.TcDUT, typeStationLocks.TcDUT, typeStationMode.TcDUT, typeStationTask.TcDUT
//   / GlobalTextList.TcGTLO, PlcTask.TcTTO, Visualization Manager.TcVMO (not stored)
//   PLC/FBs/Drives/ driveGlobals.TcGVL (not stored), driveTestCall.TcPOU (not stored), FB_DriveInterface.TcPOU (not stored), FB_DriveMotion.TcPOU (not stored)
//   PLC/FBs/FBs/Motions/ FB_Motion1way.TcPOU (not stored), FB_Motion2way.TcPOU (not stored)
//   PLC/Machine/Base/Axis/ Axis.TcGVL (not stored), AxisRowText.TcTLO (not stored), pouAxis.TcPOU (not stored)
//   PLC/Machine/Base/Axis/RowAxis/ Ax_01_AxisIncrementSelect_04.TcPOU (not stored), Ax_01_AxisMoveAbsRel_06.TcPOU (not stored), Ax_01_AxisMoveJog_05.TcPOU (not stored), Ax_01_AxisMoveTypeSelect_02.TcPOU (not stored), Ax_01_AxisNameSelect_01.TcPOU (not stored), Ax_01_AxisSpeedSelect_03.TcPOU (not stored)
//   PLC/Machine/Base/Messages/Alarms/ pouMcAlarms.TcPOU (not stored)
//   PLC/Machine/Base/Messages/ pouMsgMc.TcPOU (not stored)
//   PLC/Machine/Base/Messages/Prompts/ pouMcPrompts.TcPOU (not stored)
//   PLC/Machine/Base/Messages/Warnings/ pouMcWarnings.TcPOU (not stored)
//   PLC/Machine/Base/Station Status/ AnyStationAlarmList.TcTLO (not stored), AnyStationWarningList.TcTLO (not stored), prgAfterStationScan.TcPOU (not stored), StationNames.TcTLO (not stored)
//   PLC/Machine/Base/Units/ Mc_01_Units_02.TcPOU (not stored), Mc_01_Units_03.TcPOU (not stored), Mc_01_Units_04.TcPOU (not stored), Mc_01_Units_05.TcPOU (not stored), Mc_01_Units_06.TcPOU (not stored), pouStationUnits.TcPOU (not stored), Mc_01_Units_01.TcPOU (not stored)
//   PLC/Machine/Base/Language/ Mc_02_Language_01.TcPOU (not stored), Mc_02_Language_02.TcPOU (not stored), Mc_02_Language_03.TcPOU (not stored), Mc_02_Language_04.TcPOU (not stored), Mc_02_Language_05.TcPOU (not stored), Mc_02_Language_06.TcPOU (not stored), pouStationLangauge.TcPOU (not stored)
//   PLC/Machine/ GlobalMessages.TcGVL, Remote.TcGVL, System.TcGVL
//   PLC/Machine/Station 2/Messages/Alarms/ pouS2Alarms.TcPOU (not stored)
//   PLC/Machine/Station 2/Messages/ pouMsgS2.TcPOU (not stored)
//   PLC/Machine/Station 2/Messages/Prompts/ pouS2Prompts.TcPOU (not stored)
//   PLC/Machine/Station 2/Messages/Warnings/ pouS2Warnings.TcPOU (not stored)
//   PLC/Machine/Station 2/ pouStation2.TcPOU (not stored), S2_Global.TcGVL (not stored), S2_IO.TcGVL (not stored)
//   PLC/Machine/Station 3/Messages/Alarms/ pouS3Alarms.TcPOU (not stored)
//   PLC/Machine/Station 3/Messages/ pouMsgS3.TcPOU (not stored)
//   PLC/Machine/Station 3/Messages/Prompts/ pouS3Prompts.TcPOU (not stored)
//   PLC/Machine/Station 3/Messages/Warnings/ pouS3Warnings.TcPOU (not stored)
//   PLC/Machine/Station 3/ pouStation3.TcPOU (not stored), S3_Global.TcGVL (not stored), S3_IO.TcGVL (not stored)
//   PLC/Machine/Station 4/Messages/Alarms/ pouS4Alarms.TcPOU (not stored)
//   PLC/Machine/Station 4/Messages/ pouMsgS4.TcPOU (not stored)
//   PLC/Machine/Station 4/Messages/Prompts/ pouS4Prompts.TcPOU (not stored)
//   PLC/Machine/Station 4/Messages/Warnings/ pouS4Warnings.TcPOU (not stored)
//   PLC/Machine/Station 4/ pouStation4.TcPOU (not stored), S4_Global.TcGVL (not stored), S4_IO.TcGVL (not stored)
//   PLC/Machine/Station 5/Messages/Alarms/ pouS5Alarms.TcPOU (not stored)
//   PLC/Machine/Station 5/Messages/ pouMsgS5.TcPOU (not stored)
//   PLC/Machine/Station 5/Messages/Prompts/ pouS5Prompts.TcPOU (not stored)
//   PLC/Machine/Station 5/Messages/Warnings/ pouS5Warnings.TcPOU (not stored)
//   PLC/Machine/Station 5/ pouStation5.TcPOU (not stored), S5_Global.TcGVL (not stored), S5_IO.TcGVL (not stored)
//   PLC/Machine/Station 6/Messages/Alarms/ pouS6Alarms.TcPOU (not stored)
//   PLC/Machine/Station 6/Messages/ pouMsgS6.TcPOU (not stored)
//   PLC/Machine/Station 6/Messages/Prompts/ pouS6Prompts.TcPOU (not stored)
//   PLC/Machine/Station 6/Messages/Warnings/ pouS6Warnings.TcPOU (not stored)
//   PLC/Machine/Station 6/ pouStation6.TcPOU (not stored), S6_Global.TcGVL (not stored), S6_IO.TcGVL (not stored)
//   PLC/Machine/Station 1/ S1_IO.TcGVL (not stored), pouStation1.TcPOU (not stored), S1_Global.TcGVL (not stored)
//   PLC/Machine/Station 1/Messages/Alarms/ pouS1Alarms.TcPOU (not stored)
//   PLC/Machine/Station 1/Messages/ pouMsgS1.TcPOU (not stored)
//   PLC/Machine/Station 1/Messages/Prompts/ pouS1Prompts.TcPOU (not stored)
//   PLC/Machine/Station 1/Messages/Warnings/ pouS1Warnings.TcPOU (not stored)
//   PLC/ MAIN.TcPOU
//   X_DUTs/Tasks/ Tasks.TcGVL, TaskState.TcDUT
//   X_Language Text/Messages/Machine/ Mc_Alarms.TcTLO (not stored), Mc_Prompts.TcTLO (not stored), Mc_Warnings.TcTLO (not stored)
//   X_Language Text/Messages/Station 1/ S1_Alarms.TcTLO (not stored), S1_Prompts.TcTLO (not stored), S1_Warnings.TcTLO (not stored)
//   X_Language Text/Messages/Station 2/ S2_Alarms.TcTLO (not stored), S2_Prompts.TcTLO (not stored), S2_Warnings.TcTLO (not stored)
//   X_Language Text/Messages/Station 3/ S3_Alarms.TcTLO (not stored), S3_Prompts.TcTLO (not stored), S3_Warnings.TcTLO (not stored)
//   X_Language Text/Messages/Station 4/ S4_Alarms.TcTLO (not stored), S4_Prompts.TcTLO (not stored), S4_Warnings.TcTLO (not stored)
//   X_Language Text/Messages/Station 5/ S5_Alarms.TcTLO (not stored), S5_Prompts.TcTLO (not stored), S5_Warnings.TcTLO (not stored)
//   X_Language Text/Messages/Station 6/ S6_Alarms.TcTLO (not stored), S6_Prompts.TcTLO (not stored), S6_Warnings.TcTLO (not stored)
//   X_Sim/ FB_SimMotion.TcPOU

CONFIGURATION PLC1
    RESOURCE PLC ON TwinCAT3
        TASK DataGrab_1(INTERVAL := T#1ms, PRIORITY := 4);
        TASK PlcTask(INTERVAL := T#10ms, PRIORITY := 14);
        PROGRAM taskDataGrab WITH DataGrab_1 : taskDataGrab;
        PROGRAM MAIN WITH PlcTask : MAIN;
    END_RESOURCE
END_CONFIGURATION

// ---- Data Collection/dataAnalyse/E_BoxResultCode.TcDUT
{attribute 'qualified_only'}
{attribute 'strict'}
TYPE E_BoxResultCode :
(
    Success                     := 0,  // Signal perfectly trapped inside the box
    Err_NeverEnteredBox         := 10, // Dataset finished, signal never entered the box boundaries
    Err_IllegalEntry_SideA      := 11, // Crossed Side A (Left) but it was configured as illegal
    Err_IllegalEntry_SideC      := 13, // Crossed Side C (Top) but it was configured as illegal
    Err_IllegalEntry_SideD      := 14, // Crossed Side D (Bottom) but it was configured as illegal
	Err_WrongEntryWall			:= 15, // Entered the wrong wall!
    
    Leak_Exited_SideA           := 21, // Signal backed out of Side A (Left Wall)
    Leak_Exited_SideB           := 22, // Signal broke out of Side B (Right Wall)
    Leak_Exited_SideC           := 23, // Signal spiked over the roof out of Side C (Top Wall)
    Leak_Exited_SideD           := 24, // Signal dropped out of the floor through Side D (Bottom Wall)
    
    Violation_Exited_SideA     := 31, // Signal left Side A which was explicitly locked via IsNotPermittedToExit
    Violation_Exited_SideB     := 32, // Signal left Side B which was explicitly locked via IsNotPermittedToExit
    Violation_Exited_SideC     := 33, // Signal left Side C which was explicitly locked via IsNotPermittedToExit
    Violation_Exited_SideD     := 34  // Signal left Side D which was explicitly locked via IsNotPermittedToExit

) INT;
END_TYPE

// ---- Data Collection/dataAnalyse/E_WallEntryRule.TcDUT
// ENUM to define entry wall strictness
TYPE E_WallEntryRule :
(
    NoCheck      := 0, // Anyone can enter here. Doesn't force or block data.
    MustEnter    := 1, // Trajectory MUST enter here. If it enters somewhere else first, it fails.
    MustNotEnter := 2  // Strict wall blocker. If trajectory touches this wall, it fails immediately.
) BYTE;
END_TYPE

// ---- Data Collection/dataAnalyse/ST_BoxCorner.TcDUT
TYPE ST_BoxCorner : 
	STRUCT 
		PointXTime : LREAL; 
		PointYValue : LREAL; 
	END_STRUCT
END_TYPE

// ---- Data Collection/dataAnalyse/ST_WallPermission.TcDUT
// The updated wall permission structure
TYPE ST_WallPermission :
STRUCT
    EntryRule            : E_WallEntryRule; // Rule type: NoCheck, MustEnter, or MustNotEnter
    IsNotPermittedToExit  : BOOL;           // TRUE if not permitted to exit
END_STRUCT
END_TYPE

// ---- Data Collection/dynamicBox/structBoxData.TcDUT
TYPE structBoxData :
STRUCT
	topStatus:ST_WallPermission;
	bottomStatus:ST_WallPermission;
	leftStatus:ST_WallPermission;
	rightStatus:ST_WallPermission;
	
	topStatusChange:BOOL;
	bottomStatusChange:BOOL;
	leftStatusChange:BOOL;
	rightStatusChange:BOOL;
	
	
	    // Corner Points
    i1 : ST_BoxCorner; // Top-Left
    i2 : ST_BoxCorner; // Bottom-Left
    i3 : ST_BoxCorner; // Bottom-Right
    i4 : ST_BoxCorner; // Top-Right
	
END_STRUCT
END_TYPE

// ---- Data Collection/structAnalysis.TcDUT
TYPE structAnalysis :
STRUCT
	axis:typeDataAxis; //the data itself
	box1:structBoxData;
	box2:structBoxData;
	box3:structBoxData;
END_STRUCT
END_TYPE

// ---- Data Collection/task/typePoints.TcDUT
TYPE typePoints :
STRUCT
	PointXTime:ULINT;
	PointYValue:REAL;
END_STRUCT
END_TYPE

// ---- Data Collection/typeDataAxis.TcDUT
TYPE typeDataAxis :
STRUCT
	grabTime: ARRAY[1..20000] OF ULINT;
	grabData: ARRAY[1..20000] OF REAL;
	
END_STRUCT
END_TYPE

// ---- Data Collection/typeVectorOptions.TcDUT
TYPE typeVectorOptions :
STRUCT
	penetrateInTo:BOOL; //the line passes into the vector, into the cube
	EscapesFrom:BOOL; //the line escapes from the vector, from the cube
	DoesNotTouch:BOOL; //the line does not touch the vector
	
	point1:typePoints; //100, 60 
	point2:typePoints; //100, 40
	
	
END_STRUCT
END_TYPE

// ---- HMI1/Data/TOAST-HMI/structHMI.TcDUT
TYPE structHMI :
STRUCT
//station selected as BOOL
	gStationSelected: ARRAY[1..gHMIDataConst.gNumberOfStations] OF BOOL;
	
	//hide display elements
	gHideDisplayElements:ARRAY[0..gHMIDataConst.gNumberOfStations] OF BOOL;
	
	//stations enabled
	gStationEnabled: ARRAY[1..gHMIDataConst.gNumberOfStations] OF BOOL;
	
	gRowElementOffset: ARRAY[1..gHMIDataConst.gNumberRowsPerPage] OF UINT;
	
	//number of the active station for message display
	gNumActivePromptTextList:ARRAY[0..gHMIDataConst.gNumberOfStations] OF UINT;
	gNumActiveWarningTextList:ARRAY[0..gHMIDataConst.gNumberOfStations] OF UINT;
	gNumActiveAlarmTextList:ARRAY[0..gHMIDataConst.gNumberOfStations] OF UINT;
	
	//station selected as integer
	gActiveStationNumber:UINT; 
	
	gActivePageNumber:UINT; //current page number
	gMaxPageNumber:UINT;  //max pages exist for station, e.g. 5
	
	gActiveScreen:UINT; //combo of station + page, expressed as integer 0-999999+, reference to the text list
	
	//machine prompt number to display (summation)
	gMachinePromptNumber: UINT;

	//current number of screen on HMI
	gScreenNumber: UINT;

	//hide display elements based on what station is selected
	gHideDisplayElementAlarmView: typeStationEnables;
	gHideDisplayElementWarningView: typeStationEnables;
	gHideDisplayElementPromptView: typeStationEnables;
	
	
	gAlarmViewMsg: typeMessageRowsArry; //connect data to the HMI
	
	//header data
	hmiHeader:typeHMIheader;
	
	//language screen
	gLangRowElementOffset: ARRAY[1..gHMIDataConst.gNumberRowsPerPage] OF UINT; //seperate calculation for languages
	gLangRows: typeMotionScreen;
	gLangButtons: typeMotionScreenBtn;
	gActiveLangPageNumber:UINT; //current page number for units
	gMaxPageNumberLang:UINT;  //max pages exist for station, e.g. 5
	
	gHMIScreenString:STRING;
	
	//title of manual motion screen
	gManualScreenTitle:UINT;
	
	gVisuHasInited:BOOL;
	
	//buttons to lock a station
	gStateLockStation1: USINT;
	gStateLockStation2: USINT;
	gStateLockStation3: USINT;
	gStateLockStation4: USINT;
	gStateLockStation5: USINT;
	gStateLockStation6: USINT;
	
END_STRUCT
END_TYPE

// ---- HMI1/Data/TOAST-HMI/structHMIBtns.TcDUT
TYPE structHMIBtns :
STRUCT
	//buttons to select a station
	btnSelectStation1: BOOL;
	btnSelectStation2: BOOL;
	btnSelectStation3: BOOL;
	btnSelectStation4: BOOL;
	btnSelectStation5: BOOL;
	btnSelectStation6: BOOL;

	btnSelectAll: BOOL;	//button to select all stations
	btnAllStationsSelected: BOOL;

	//reset button for global use
	btnReset: BOOL;

	//manual screen
	btnAbsMode:BOOL; //TRUE if abs mode, False if sys mode
	btnNextPage: BOOL;
	btnPrevPage: BOOL;
	
	//hide button data for main screen
	btnHides:typeBtnHides;
	
	//hmi buttons
	btnMode:typeBtnPress;
	
	//hmi buttons feedback
	btnFdbk: typeBtnFdbk;
	
	btnPlus1Row:BOOL; //scroll 1 row up
	btnNeg1Row:BOOL; //scroll 1 row down
	clk: INT;
	
	gAnyButtonPressed:BOOL; //TRUE if any button was pressed
	
		//buttons to lock a station
	btnLockStation1: BOOL;
	btnLockStation2: BOOL;
	btnLockStation3: BOOL;
	btnLockStation4: BOOL;
	btnLockStation5: BOOL;
	btnLockStation6: BOOL;
	
	gLockButtons:typeStationLockModes;
	
END_STRUCT
END_TYPE

// ---- HMI1/Data/TOAST-HMI/structHMIGlobal.TcDUT
TYPE structHMIGlobal :
STRUCT
	hmi:structHMI;
	btns:structHMIBtns;
	GlobalMessages:structHMIMessages;
	
END_STRUCT
END_TYPE

// ---- HMI1/Data/TOAST-HMI/structHMIMessages.TcDUT
TYPE structHMIMessages :
STRUCT
		//define messages for machine base
	gMsgMc	:typeStationMessage;
	
	//define message for each station
	gMsgS1	:typeStationMessage;
	gMsgS2	:typeStationMessage;
	gMsgS3	:typeStationMessage;
	gMsgS4	:typeStationMessage;
	gMsgS5	:typeStationMessage;
	gMsgS6	:typeStationMessage;
	
	//global memory for retaining status of station
	gMsgMcStat	:typeStationStatus;
	gMsgS1Stat	:typeStationStatus;
	gMsgS2Stat	:typeStationStatus;
	gMsgS3Stat	:typeStationStatus;
	gMsgS4Stat	:typeStationStatus;
	gMsgS5Stat	:typeStationStatus;
	gMsgS6Stat	:typeStationStatus;
	
	//list view of messages in array form
	gListMsgMc	:typeMessageRowsArry;
	gListMsgS1	:typeMessageRowsArry;
	gListMsgS2	:typeMessageRowsArry;
	gListMsgS3	:typeMessageRowsArry;
	gListMsgS4	:typeMessageRowsArry;
	gListMsgS5	:typeMessageRowsArry;
	gListMsgS6	:typeMessageRowsArry;

	gAnyFaultMessage: BOOL; //TRUE if there are any fault messages (any)
	gAnyWarnings: BOOL; //TRUE if there are any warnings (the yellow ones)

	//alarm view of messages in alarmview form
	gMcAlarmView: typeAlarmViewStation;
	gS1AlarmView: typeAlarmViewStation;
	gS2AlarmView: typeAlarmViewStation;
	gS3AlarmView: typeAlarmViewStation;
	gS4AlarmView: typeAlarmViewStation;
	gS5AlarmView: typeAlarmViewStation;
	gS6AlarmView: typeAlarmViewStation;
	
	gHMIAlarmView: typeAlarmViewStation;
END_STRUCT
END_TYPE

// ---- HMI1/Screens/Machine Settings/typeRecord.TcDUT
TYPE typeRecord :
STRUCT
	sName 	: T_MaxString 	:= '';
	nNumber	: UDINT 		:= 0;
	fPos	: LREAL 		:= 0.0;
	bOP		: BOOL 			:= FALSE;
	sDesc	: STRING(40)	:= '';
	data	: ARRAY[0..7] OF BYTE;
END_STRUCT
END_TYPE

// ---- HMI1/Screens/Machine Settings/typeSettings.TcDUT
TYPE typeSettings :
	STRUCT
		TextName:STRING := ('Unnamed Setting');
		Value:INT;
		hasChanged:BOOL;
	END_STRUCT
END_TYPE

// ---- PLC/Safety/enumEstopState.TcDUT
{attribute 'qualified_only'}
{attribute 'strict'}

//TwinSAFE-Logic-FBen.pdf
//Table 3-24: State information (8-bit value)

TYPE enumEstopState :
(
	undefined	:=	0,
	Run			:=	1,
	Stop		:=	2,
	Safe		:=	3,
	Error		:=	4,
	Reset		:=	5,
	Start		:=	6,
	NoStateDef1	:=	7,
	DelayOut	:=	8,
	NoStateDef2	:=	9
);
END_TYPE

// ---- PLC/Safety/structEstopDiag.TcDUT
TYPE structEstopDiag :
UNION
	iwordvalue:UINT;
	bitvalue:structSafetyEstopDiagBOOList;
END_UNION
END_TYPE

// ---- PLC/Safety/structSafetyEstopDiagBOOList.TcDUT
TYPE structSafetyEstopDiagBOOList :
STRUCT
	//from Function blocks for TwinSAFE logic components.pdf
	//3.4.2.1 Diagnostic and state information for FB ESTOP
	b0_DiscrapencyErrorInputGroup1	:BOOL;
	b1_DiscrapencyErrorInputGroup2	:BOOL;
	b2_DiscrapencyErrorInputGroup3	:BOOL;
	b3_DiscrapencyErrorInputGroup4	:BOOL;
	b4_EDMmonitoringErrorEDM1		:BOOL;
	b5_EDMmonitoringErrorEDM2		:BOOL;
	b6_NotUsed						:BOOL;
	b7_NotUsed						:BOOL;
	b8_DiscrepancyErrorInputGroup1	:BOOL; //with activated option "Safe Inputs after Disc Error" 
	b9_DiscrepancyErrorInputGroup2	:BOOL; //with activated option "Safe Inputs after Disc Error"
	b10_DiscrepancyErrorInputGroup3	:BOOL; //with activated option "Safe Inputs after Disc Error"
	b11_DiscrepancyErrorInputGroup4	:BOOL; //with activated option "Safe Inputs after Disc Error"
	b12_NotUsed						:BOOL; 
	b13_NotUsed						:BOOL; 
	b14_NotUsed						:BOOL; 
	b15_NotUsed						:BOOL;  
END_STRUCT
END_TYPE

// ---- X_DUTs/Diagnostic/typeDPSlaveIndicator.TcDUT
TYPE typeDPSlaveIndicator :
STRUCT
	currentState:DWORD; //inside colour
	historicalState:DWORD; //outside colour
	SlaveNumber:UINT; //slave number 1-127
END_STRUCT
END_TYPE

// ---- X_DUTs/Diagnostic/typeEtherCATIndicator.TcDUT
TYPE typeEtherCATIndicator :
STRUCT
	currentState:typeEtherCATState; //inside colour
	historicalState:typeEtherCATState; //outside colour
	SlaveNumber:UINT; //slave number 1-65535
	isPresent: BOOL; //TRUE if node is present in config
	
	//extra diagnostics
	ConfigData:ST_EcSlaveConfigData;
	crcCount:ST_EcCrcError;
	
	//PLC ordering number
	hmiNum:UINT;
END_STRUCT
END_TYPE

// ---- X_DUTs/Diagnostic/typeEtherCATmasters.TcDUT
TYPE typeEtherCATmasters :
STRUCT
	ecAMSmaster AT %I* :AMSNETID;
	//ecAMSbytesmaster: T_AmsNetIdArr;
	ecAMSmasterstr: T_AmsNetID;
	ecMasterCfgSlaveCount AT %I* : UINT;
	ecMasterActSlaveCount AT %I* : UINT;
	ecMasterDevId AT %I* : UINT;
	ecMasterChangeCount AT %I* : UINT;
	ecMasterDevState AT %I* : UINT;
	ecEKInfostateDataState AT %I* : UINT;
END_STRUCT
END_TYPE

// ---- X_DUTs/Diagnostic/typeEtherCATState.TcDUT
TYPE typeEtherCATState :
STRUCT
	//suffix code
	//0x___1 = Slave in 'INIT' state
	//0x___2 = Slave in 'PREOP' state
	//0x___3 = Slave in 'BOOT' state
	//0x___4 = Slave in 'SAFEOP' state
	//0x___8 = Slave in 'OP' state
	state:EtherCATstate;

	
	
	//prefix code
	//0x001_ = Slave signals error
	//0x002_ = Invalid vendorId, productCode... read
	//0x004_ = Initialization error occurred
	//0x008_ = Slave disabled
	//0x010_ = Slave not present
	//0x020_ = Slave signals link error
	//0x040_ = Slave signals missing link
	//0x080_ = Slave signals unexpected link
	//0x100_ = Communication port A
	//0x200_ = Communication port B
	//0x400_ = Communication port C
	//0x800_ = Communication port D
	suffix:EtherCATSuffix;
	
	isFault:BOOL; //TRUE if either state is not 8 and code exists
	colour:DWORD; //colour state
	
	

END_STRUCT
END_TYPE

// ---- X_DUTs/Diagnostic/typePROFINETIndicator.TcDUT
TYPE typePROFINETIndicator :
STRUCT
	currentState:typeProfiNetState; //inside colour
	historicalState:typeProfiNetState; //outside colour
	SlaveNumber:UINT; //slave number 1-65535
	isPresent: BOOL; //TRUE if node is present in config
	
	//extra diagnostics
	//tbd
END_STRUCT
END_TYPE

// ---- X_DUTs/Diagnostic/typeProfiNetMaster.TcDUT
TYPE typeProfiNetMaster :
STRUCT
	
DevState:UINT;
//0x0001 = No link AT port 1
//0x0002 = No link at port 2
//0x0010 = Out of send resources (I/O reset required)
//0x0080 = I/O reset active





PnIoError:UINT;
//Error:indicates the number of PnIo boxes with a error



PnIoDiag:UINT;
//Warning:indicates the number of PnIo boxes with a warning or diagnosis




END_STRUCT
END_TYPE

// ---- X_DUTs/Diagnostic/typePROFINETState.TcDUT
TYPE typePROFINETState :
STRUCT
	//PnIoBoxState
	//UINT
	//0 = No error
	//1 = Profinet device state machine is in boot mode
	//2 = Device not found
	//3 = The stationname is not unique
	//4 = IP could not be set
	//5 = IP conflict
	//6 = DCP set was not successful
	//7 = Watchdog error
	//8 = Datahold error
	//9 = RTC3: Sync mode could not be initiated
	//10 = Profinet controller has a link error
	//11 = The aliasname is not unique
	//12 = The automatic name assignement isn't possible - wrong device type
	//13 = IOC-AR is established but no application ready
	//14 = IOC-AR is established but module difference
	//15 = At least one InputCR is invalid, provider in stop or problemindicator is set
	//16 = At least one OutputCR is invalid, provider in stop or problemindicator is set
	//31 = Only for EtherCAT gateways: WC-State of cyclic EtherCAT frame is 1

	state:ProfiNetstate;

	
	
	//PnIoBoxDiag
	//UINT
	//0x0000 = No diagnosis
	//0x0001 = IOC-AR is not established
	//0x0002 = IOC-AR is established
	//0x0004 = IOC-AR is established but no application ready
	//0x0008 = IOC-AR is established but module difference
	//0x0010 = At least one AlarmCR got a diagnosis alarm
	//0x0100 = At least one InputCR is invalid
	//0x0200 = At least one InputCR Provider is in stop
	//0x0400 = At least one InputCR Problemindicator is set
	//0x1000 = At least one OutputCR is invalid
	//0x2000 = At least one OutputCR Provider is in stop
	//0x4000 = At least one OutputCR Problemindicator is set

	suffix:ProfiNetSuffix;
	
	isFault:BOOL; //TRUE if either state is not 8 and code exists
	colour:DWORD; //colour state
	
	

END_STRUCT
END_TYPE

// ---- X_DUTs/Drives/HMIaxisDefinition.TcDUT
TYPE HMIaxisDefinition :
STRUCT
	//define axis type for display on HMI. Does not affect axis_ref
	AxisName: STRING:='Linear Slide';
	AxisDef: STRING :='X';
	AxisNumber: int;
	isLinearDrive: BOOL; //TRUE if the drive exists as a linear position in mm
	isSpindleDrive: BOOL; //TRUE if the drive is a spindle



END_STRUCT
END_TYPE

// ---- X_DUTs/Drives/typeDriveInterface.TcDUT
TYPE typeDriveInterface :
STRUCT
	//logic to run
	enableAxis: BOOL; //TRUE to enable the axis
	isDriveBusy: BOOL; //TRUE if the drive is doing something
	generalResetReq: BOOL; //TRUE to reset command to the drives
	isAbsMove: BOOL; //TRUE if abs move
	isRelMove: BOOL; //TRUE if rel move
	MoveReq: BOOL; //TRUE to move the drive
	isManualMode: BOOL; //TRUE to run a lower speeds

	isVeloMove:BOOL; //TRUE if velocity move
	veloDirection:MC_Direction; //direction of velocity
	
	
	
	//speeds and feeds
	TargetPosn: LREAL;
	TargetVelo: LREAL;
	TargetAcc:LREAL;
	TargetDec:LREAL;
	TargetJerk:LREAL;
	
	//feedback value from drive
	actualPosn:LREAL;
	actualVelo:LREAL;
	
	//set posn
	SetPosn:BOOL; //TRUE to set new posn
	newPosn:LREAL; //new posn target

	//error word feedback
	AxisErrorID : DWORD;
	
	jogFwdReq:BOOL; //TRUE to jog forward
	jogRevReq:BOOL; //TRUE to jog reverse
	
	


END_STRUCT
END_TYPE

// ---- X_DUTs/HMI/typeBtnFdbk.TcDUT
TYPE typeBtnFdbk :
STRUCT
	
//button Fdbk BOOLs for mode screen

////	|------------------------------------|
////	|									 |
////	|a	00 01 02 03 04 05 06 07 08 09	x|
////	|b	10 11 12 13 14 15 16 17 18 19	y|
//// 	|   20 21 22 23 24 25 26 27 28 29	 |
//// 	|   30 31 32 33 34 35 36 37 38 39	 |
////	|									 |
////	|									 |
////	|------------------------------------|

//button Fdbk BOOL in X-Y format
//a,b,x,y are not included
//a,b are power on / off, these never get hidden
//x,y are auto cycle start, these normally dont get hidden
	btn00Fdbk: BOOL;
	btn01Fdbk: BOOL;
	btn02Fdbk: BOOL;
	btn03Fdbk: BOOL;
	btn04Fdbk: BOOL;
	btn05Fdbk: BOOL;
	btn06Fdbk: BOOL;
	btn07Fdbk: BOOL;
	btn08Fdbk: BOOL;
	btn09Fdbk: BOOL;

	btn10Fdbk: BOOL;
	btn11Fdbk: BOOL;
	btn12Fdbk: BOOL;
	btn13Fdbk: BOOL;
	btn14Fdbk: BOOL;
	btn15Fdbk: BOOL;
	btn16Fdbk: BOOL;
	btn17Fdbk: BOOL;
	btn18Fdbk: BOOL;
	btn19Fdbk: BOOL;
	
	btn20Fdbk: BOOL;
	btn21Fdbk: BOOL;
	btn22Fdbk: BOOL;
	btn23Fdbk: BOOL;
	btn24Fdbk: BOOL;
	btn25Fdbk: BOOL;
	btn26Fdbk: BOOL;
	btn27Fdbk: BOOL;
	btn28Fdbk: BOOL;
	btn29Fdbk: BOOL;
	
	//btn30Fdbk: BOOL;
	//btn31Fdbk: BOOL;
	//btn32Fdbk: BOOL;
	//btn33Fdbk: BOOL;
	//btn34Fdbk: BOOL;
	//btn35Fdbk: BOOL;
	//btn36Fdbk: BOOL;
	//btn37Fdbk: BOOL;
	//btn38Fdbk: BOOL;
	//btn39Fdbk: BOOL;

	btnAutoCyclingFdbk: BOOL; //auto cycling for station
	btnIsHomeFdbk: BOOL;	//TRUE if station is at home
	btnIsSEOCFdbk:BOOL;		//TRUE if the station is SEOC'in
	btnControlFdbk:BOOL;	//TRUE if the station is under control, for use cases of multiple Visu's
	btnModeFdbk:BOOL;


END_STRUCT
END_TYPE

// ---- X_DUTs/HMI/typeBtnHides.TcDUT
TYPE typeBtnHides :
STRUCT
	
//button hide BOOLs for mode screen

////	|------------------------------------|
////	|									 |
////	|a	00 01 02 03 04 05 06 07 08 09	x|
////	|b	10 11 12 13 14 15 16 17 18 19	y|
//// 	|   20 21 22 23 24 25 26 27 28 29	 |
//// 	|   30 31 32 33 34 35 36 37 38 39	 |
////	|									 |
////	|									 |
////	|------------------------------------|

//button hide BOOL in X-Y format
//a,b,x,y are not included
//a,b are power on / off, these never get hidden
//x,y are auto cycle start, these normally dont get hidden
	btn00Hide: BOOL;
	btn01Hide: BOOL;
	btn02Hide: BOOL;
	btn03Hide: BOOL;
	btn04Hide: BOOL;
	btn05Hide: BOOL;
	btn06Hide: BOOL;
	btn07Hide: BOOL;
	btn08Hide: BOOL;
	btn09Hide: BOOL;

	btn10Hide: BOOL;
	btn11Hide: BOOL;
	btn12Hide: BOOL;
	btn13Hide: BOOL;
	btn14Hide: BOOL;
	btn15Hide: BOOL;
	btn16Hide: BOOL;
	btn17Hide: BOOL;
	btn18Hide: BOOL;
	btn19Hide: BOOL;
	
	btn20Hide: BOOL;
	btn21Hide: BOOL;
	btn22Hide: BOOL;
	btn23Hide: BOOL;
	btn24Hide: BOOL;
	btn25Hide: BOOL;
	btn26Hide: BOOL;
	btn27Hide: BOOL;
	btn28Hide: BOOL;
	btn29Hide: BOOL;
	
	btn30Hide: BOOL;
	btn31Hide: BOOL;
	btn32Hide: BOOL;
	btn33Hide: BOOL;
	btn34Hide: BOOL;
	btn35Hide: BOOL;
	btn36Hide: BOOL;
	btn37Hide: BOOL;
	btn38Hide: BOOL;
	btn39Hide: BOOL;


END_STRUCT
END_TYPE

// ---- X_DUTs/HMI/typeBtnPress.TcDUT
TYPE typeBtnPress :
STRUCT
	
//button Pressed BOOLs for mode screen

////	|------------------------------------|
////	|									 |
////	|a	00 01 02 03 04 05 06 07 08 09	x|
////	|b	10 11 12 13 14 15 16 17 18 19	y|
//// 	|   20 21 22 23 24 25 26 27 28 29	 |
//// 	|   30 31 32 33 34 35 36 37 38 39	 |
////	|									 |
////	|									 |
////	|------------------------------------|

//button Pressed BOOL in X-Y format
//a,b,x,y are not included
	btn00Pressed: BOOL;
	btn01Pressed: BOOL;
	btn02Pressed: BOOL;
	btn03Pressed: BOOL;
	btn04Pressed: BOOL;
	btn05Pressed: BOOL;
	btn06Pressed: BOOL;
	btn07Pressed: BOOL;
	btn08Pressed: BOOL;
	btn09Pressed: BOOL;

	btn10Pressed: BOOL;
	btn11Pressed: BOOL;
	btn12Pressed: BOOL;
	btn13Pressed: BOOL;
	btn14Pressed: BOOL;
	btn15Pressed: BOOL;
	btn16Pressed: BOOL;
	btn17Pressed: BOOL;
	btn18Pressed: BOOL;
	btn19Pressed: BOOL;
	
	btn20Pressed: BOOL; //gate 1 access request
	btn21Pressed: BOOL; //gate 2 access request
	btn22Pressed: BOOL; //gate request cancel
	btn23Pressed: BOOL;
	btn24Pressed: BOOL;
	btn25Pressed: BOOL;
	btn26Pressed: BOOL;
	btn27Pressed: BOOL;
	btn28Pressed: BOOL;
	btn29Pressed: BOOL;
	
	//btn30Pressed: BOOL;
	//btn31Pressed: BOOL;
	//btn32Pressed: BOOL;
	//btn33Pressed: BOOL;
	//btn34Pressed: BOOL;
	//btn35Pressed: BOOL;
	//btn36Pressed: BOOL;
	//btn37Pressed: BOOL;
	//btn38Pressed: BOOL;
	//btn39Pressed: BOOL;

	//special case buttons	
	btnPowerOnPressed: BOOL; //TRUE to power the machine on
	btnPowerOffPressed: BOOL; //TRUE to power the machine off

	btnAutoCycleStartPressed: BOOL; //TRUE to start auto cycle
	btnAutoCycleStopPressed: BOOL; //TRUE to stop auto cycle immediately

	btnFooterAutoCycleStart: BOOL;
	btnFooterAutoCycleStopEOC: BOOL;
	btnFooterReturnHome: BOOL;
	btnFooterAutoMode: BOOL;
	btnFooterManualMode: BOOL;




END_STRUCT
END_TYPE

// ---- X_DUTs/HMI/typeHMIheader.TcDUT
TYPE typeHMIheader :
STRUCT
	
	stationstate: INT;
	stationstateColour:BOOL;
	homestate: INT; //home state for text list
	homestateColour: BOOL; //colour state of indicator

	anotherstate: BOOL;
	//faultstate: BOOL;
	//stationname: BOOL;
	flasher: BOOL;

	stationNameSelect: UINT; //station name selection
	cycleTypeFeedback: INT;
	
	isFaultState: BOOL; //colour change header
	FaultStateHeader: INT; //text change on header
	
	AnyStationFaultHeaderActive:BOOL;//colour change for global header
	AnyStationFaultHeader:INT; //text select for global header
	AnyStationFaultColour:DWORD; //background blue, alarm red or warning yellow
	isAnyFaultState: BOOL; //colour change header
	
	isWarningState: BOOL; //colour change header
	WarningStateHeader: INT; //text change on header
	
	AnyStationWarningHeaderActive:BOOL;//colour change for global header
	AnyStationWarningHeader:INT; //text select for global header
	AnyStationWarningColour:DWORD; //background blue, alarm red or warning yellow
	isAnyWarningState: BOOL; //colour change header







END_STRUCT
END_TYPE

// ---- X_DUTs/HMI/typeMessageRowsArry.TcDUT
TYPE typeMessageRowsArry :
STRUCT
	
	AlarmViewMsg : ARRAY[1..gHMIDataConst.gNumberOfMessagesScreen] OF typeMessageRow;
	WarningViewMsg : ARRAY[1..gHMIDataConst.gNumberOfMessagesScreen] OF typeMessageRow;
	PromptViewMsg : ARRAY[1..gHMIDataConst.gNumberOfMessagesScreen] OF typeMessageRow;

END_STRUCT
END_TYPE

// ---- X_DUTs/MessageView/typeNewMsg.TcDUT
TYPE typeNewMsg :
STRUCT
	
timeRaised:STRING(12):='12:23:32';;
timeResolved:STRING(12):='13:43:12';
text:STRING(255);
source:STRING(10);


END_STRUCT
END_TYPE

// ---- X_DUTs/MessageView/typeNewMsgStyle.TcDUT
TYPE typeNewMsgStyle :
STRUCT
	
isColoured:BOOL;			//TRUE to apply a colour, e.g. RED or YELLOW, normal messages = false, so grey
colourToApply:DWORD;		//from consts in global HMIColour


END_STRUCT
END_TYPE

// ---- X_DUTs/Motion/typeMotionRecordRow.TcDUT
TYPE typeMotionRecordRow :
STRUCT
	Advanced:ULINT; //number of advanced
	Returned:ULINT; //number of returned
	stnPosnInput:STRING; //input value 
END_STRUCT
END_TYPE

// ---- X_DUTs/Motion/typeMotionRow.TcDUT
TYPE typeMotionRow :
STRUCT
	
	Advance:typeMotionSide; //advance data
	Returned:typeMotionSide; //return data
	
	strPosn:STRING; //formatted position, in string form

	IndexLocation:UINT :=10; //index value
	
	bHidePosn: BOOL; //TRUE to hide the posn
	bHideName: BOOL; //TRUE to hide the name
	
	bIsAbsSymSwitch: BOOL; //TRUE to switch between abs/symb
	
END_STRUCT
END_TYPE

// ---- X_DUTs/Motion/typeMotionRowArry.TcDUT
TYPE typeMotionRowArry :
STRUCT
	data: ARRAY[1..99] OF typeMotionRecordRow;
END_STRUCT
END_TYPE

// ---- X_DUTs/Motion/typeMotionRowButtons.TcDUT
TYPE typeMotionRowButtons :
STRUCT
	//beckhoff visu can't deal with in_out as a passed typed with both inputs and outputs, so the feedback (buttons) are passed in a seperate memory area
	btnAdvance: BOOL; //Press to advance motion
	btnReturn: BOOL; //press to return motion
	
	
	stnPosnInput:STRING; //input value 
	
END_STRUCT
END_TYPE

// ---- X_DUTs/Motion/typeMotionRowIO.TcDUT
TYPE typeMotionRowIO :
STRUCT
	
	//structure for a conventional motion (air cylinder, etc)

	iAdvanceDepth		AT %I* :BOOL;
	iReturnedDepth		AT %I* :BOOL;
	
	qAdvanceCoil		AT %Q* :BOOL;
	qReturnedCoil		AT %Q* :BOOL;
	

END_STRUCT
END_TYPE

// ---- X_DUTs/Motion/typeMotionSide.TcDUT
TYPE typeMotionSide :
STRUCT
	RequestCoil: BOOL;		//TRUE if the coil to advance the motion has been switched on
	Depth: BOOL;  			//TRUE if the motion is complete
	Prompt: BOOL;           //TRUE if the motion is OK to move (or to the next step)
	InterlockOK: BOOL;		//TRUE if the interlock is satisified for the motion
	NumberOrder:UINT;		//number of the motion to take

	TimeTaken: TIME;		//Time Taken for the motion to complete
	
	valCoil: INT := 1;		
	valDepth: INT := 2;
	
	bHideCoil: BOOL;		//TRUE to hide the coil
	bHideDepth: BOOL;		//TRUE to hide the depth
	bHideInterlock: BOOL;	//TRUE to hide the interlock
	bHidePrompt: BOOL;		//TRUE to hide the prompt
	bHideTime: BOOL;		//TRUE to hide the time
	bHideButton: BOOL;		//TRUE to hide the button
	
	FdbkColour: DWORD := 16#FFC6C6C6; //sensor feedback colour
	CoilColour:DWORD := 16#FFC6C6C6; //coil feedback colour


END_STRUCT
END_TYPE

// ---- X_DUTs/Screen/typeMotionScreen.TcDUT
TYPE typeMotionScreen :
STRUCT
	
	//define motion rows for HMI
	//define all rows that will fit on a screen for a given resolution
	//feedback from the PLC to the HMI
	gMotionRow1: typeMotionRow;
	gMotionRow2: typeMotionRow;
	gMotionRow3: typeMotionRow;
	gMotionRow4: typeMotionRow;
	gMotionRow5: typeMotionRow;
	gMotionRow6: typeMotionRow;
	gMotionRow7: typeMotionRow;
	gMotionRow8: typeMotionRow;
	gMotionRow9: typeMotionRow;

END_STRUCT
END_TYPE

// ---- X_DUTs/Screen/typeMotionScreenBtn.TcDUT
TYPE typeMotionScreenBtn :
STRUCT
	//define motion rows for HMI
	//signals from the buttons to the PLC request
	gMotionRow1btn: typeMotionRowButtons;
	gMotionRow2btn: typeMotionRowButtons;
	gMotionRow3btn: typeMotionRowButtons;
	gMotionRow4btn: typeMotionRowButtons;
	gMotionRow5btn: typeMotionRowButtons;
	gMotionRow6btn: typeMotionRowButtons;
	gMotionRow7btn: typeMotionRowButtons;
	gMotionRow8btn: typeMotionRowButtons;
	gMotionRow9btn: typeMotionRowButtons;
END_STRUCT
END_TYPE

// ---- X_DUTs/Setup/typeSetupStation.TcDUT
TYPE typeSetupStation :
STRUCT
	
	allowAutoCycle: BOOL:=TRUE;
	allowManualMode: BOOL:=TRUE;
	allowSemiAuto: BOOL:=TRUE;
	allowDryCycle: BOOL:=TRUE;
	allowBypass: BOOL:=TRUE;
	allowContinuousCycle: BOOL:=TRUE;
	allowSingleCycle: BOOL:=TRUE;
	allowSEOC: BOOL:=TRUE;
	allowPowerOn: BOOL:=TRUE;
	allowPowerOff:BOOL:=TRUE;
	allowServicesPowerOn:BOOL:=TRUE;
	allowRemoteControl:BOOL:=TRUE;
	allowSilenceHorn:BOOL:=TRUE;
	allowGate1Req:BOOL:=TRUE;
	allowGate2Req:BOOL:=TRUE;
	allowLockAccessGates:BOOL:=TRUE;
	allowEnablePendent:BOOL:=TRUE;
	
	//number of rows programmed
	numRowsConfig:USINT := 0;
	
	
	
	
	


END_STRUCT
END_TYPE

// ---- X_DUTs/Station/enumStationState.TcDUT
{attribute 'qualified_only'}
{attribute 'strict'}
TYPE enumStationState :
(
	noState			:=	0,
	Loading			:=	1,
	Cycling			:=	2,
	Unloading		:=	3,
	Spare			:=	4,
	Blocked			:=	5,
	Starved			:=	6,
	WaitAux			:=	7,
	Faulted			:=	8,
	Repair			:=	9,
	EStop			:=	10,
	Manstop			:=	11,
	Other			:=	12
	
	
);
END_TYPE

// ---- X_DUTs/Station/typeIndividualTask.TcDUT
TYPE typeIndividualTask :
STRUCT
	singleTaskName:STRING(255):='Unnamed Task';
	CycleTimeTarget: REAL :=60.0;	//target cycle time, e.g. 60s
	CycleTimeActual: REAL :=0;		//actual cycle time
	CycleTimePartOver:REAL:=5;		//cycle time is part over, e.g. 5s
	CycleTimeGrossOver:REAL:=120; 	//time for grossly over cycle time
	CycleTimeLast: REAL;			//last part cycle time
	OverCycleTime:BOOL;				//TRUE if over cycle time
	CycleTimeIsGrossOver:BOOL;		//TRUE if cycle time is grossly over
	IsTaskEnabled:BOOL;				//TRUE if the task is enabled
	IsTaskComplete:BOOL;			//TRUE if the task is complete
	TaskStatus:USINT;				//task status
	StateColour:DWORD; 				//colour state of task indicator
	
	IsTaskPassed:BOOL;				//TRUE if the task was PASSED...
	IsTaskFailed:BOOL;				//TRUE if the task was FAILED, but still complete
	IsTaskRejected:BOOL;
	IsTaskSkipped:BOOL;
	IsTaskBypassed:BOOL;
	
	complexity:UINT;				//complexity of part for task

END_STRUCT
END_TYPE

// ---- X_DUTs/Station/typeStation.TcDUT
TYPE typeStation :
STRUCT
	Data: typeStationMode;
	hmiHeader:typeHMIheader;
	
	//all motion rows in the station, to be inserted into the main HMI motion screen
	MotionRow: ARRAY[1..99] OF typeMotionRow;
	MotionRowBtn: ARRAY[1..99] OF typeMotionRowButtons;
	
	//part data
	part: typeStationTask; //part data for each station
	
	//record of motions
	MotionRecordStation: typeMotionRowArry;
	
	dynRowNumber :UINT; //dynamic row caller
END_STRUCT
END_TYPE

// ---- X_DUTs/Station/typeStationComplexity.TcDUT
TYPE typeStationComplexity :
STRUCT
	task:UINT;
	complexity:uint;
	
END_STRUCT
END_TYPE

// ---- X_DUTs/Station/typeStationComplexityBuffer.TcDUT
TYPE typeStationComplexityBuffer :
STRUCT
	buffer: ARRAY[0..2048] OF BYTE;
	
	
END_STRUCT
END_TYPE

// ---- X_DUTs/Station/typeStationLockModes.TcDUT
TYPE typeStationLockModes :
STRUCT
	btnStartAutoCycle: 		BOOL; //button to start auto cycle
	btnStopAutoCycle: 		BOOL; //button to stop auto cycle	
 
	btnReset: 				BOOL; //button to reset station
	
	btnSelectAutoMode: 		BOOL; //button to select auto mode
	btnSelectManualMode: 	BOOL; //button to select manual mode
	btnSelectSemiAutoMode: 	BOOL; //button to select semi auto mode
	btnSelectDryCycleMode: 	BOOL; //button to select dry cycle mode
	btnSelectWetCycleMode: 	BOOL; //button to select wet cycle mode (endless cycles with inserts, no part transfer to next station)
	
	btnSelectContCycleMode: 	BOOL; 
	btnSelectSingleCycleMode: 	BOOL; 
	
	btnSEOC:					BOOL;
	
	
END_STRUCT
END_TYPE

// ---- X_DUTs/Station/typeStationLocks.TcDUT
TYPE typeStationLocks :
STRUCT
	Station1Locked:BOOL;
	Station2Locked:BOOL;
	Station3Locked:BOOL;
	Station4Locked:BOOL;
	Station5Locked:BOOL;
	Station6Locked:BOOL;
						
END_STRUCT
END_TYPE

// ---- X_DUTs/Station/typeStationMode.TcDUT
TYPE typeStationMode :
STRUCT
	Manual:					BOOL :=TRUE; //TRUE if the station is in manual mode
	AutoCycle:				BOOL; //TRUE if the station is in auto mode
	AutoCycling:			BOOL; //TRUE if the station is auto cycling
	SemiAuto:				BOOL; //TRUE if the station is in semi auto (magic prompting)
	DryCycle:				BOOL; //TRUE if the station is in dry run mode (no parts)
	ModeValue:				INT;  //integer value of the mode for display
	Bypass:					BOOL; //TRUE if the station is in bypass mode (no process to be performed)
	ContCycle:				BOOL :=TRUE;
	SingleCycle:			BOOL; //TRUE if the station is in single cycle mode
	StopEOC:				BOOL; //TRUE if the station is stopping at end of cycle
	Fault:					BOOL; //TRUE if the station is in fault state
	Warning:				BOOL; //TRUE if the station is in a warning state
	CycleStopping:			BOOL; //TRUE if the cycle is stopping


	btnStartAutoCycle: 		BOOL; //button to start auto cycle
	btnStopAutoCycle: 		BOOL; //button to stop auto cycle	
 
	btnReset: 				BOOL; //button to reset station
	
	btnSelectAutoMode: 		BOOL; //button to select auto mode
	btnSelectManualMode: 	BOOL; //button to select manual mode
	btnSelectSemiAutoMode: 	BOOL; //button to select semi auto mode
	btnSelectDryCycleMode: 	BOOL; //button to select dry cycle mode
	btnSelectWetCycleMode: 	BOOL; //button to select wet cycle mode (endless cycles with inserts, no part transfer to next station)
	
	NumOfRows:				UINT; //number of motions present in station in rows CEIL by number of rows permitted in the screen
	NumOfUnitRows:			UINT; //number of motions present in station in rows CEIL by number of rows permitted in the screen
	NumOfLangRows:			UINT; //number of motions present in station in rows CEIL by number of rows permitted in the screen
	NumberOfPages:			UINT; //number of pages in the station that can fit for the number of motion rows
		
	StationNumber:			UINT; //the station number, typ. 1-6
	
	PowerOn:				BOOL; //TRUE if the machine is Powered On
	MotionPowerOn:			BOOL; //TRUE if the machine is powered on with motion, e.g. servo enable, pneumatic air on, hydraulics on,

	IsStationSelectedHMI:	BOOL; //Is the station selected on the HMI
	
	StationState:			INT; //state value as integer
	
	IsHome:					BOOL; //TRUE if the station is HOME
	IsHoming: 				BOOL; //TRUE if the station is in the process of returning to home
	IsRemote:				BOOL; //TRUE if the station is in remote mode
	
	StationStateColour:     DWORD;//colour feedback for station state of main screen
	StationStateTextColour: DWORD;//colour feedback for station state of main screen
	
	stepNum:				INT;
	stepNumListing:			ARRAY[0..32767] OF INT;
	sizeofStepListing:		INT := 32767;
	
	latchXICmsg:			BOOL :=FALSE; //TRUE to latch in XIC messages and require a reset button press to resolve, FALSE to only latch on auto XIC faults
	
	IsStationLocked:		BOOL;	//TRUE if the station is locked to other stations
	
	
	
	
	


END_STRUCT
END_TYPE

// ---- X_DUTs/Station/typeStationTask.TcDUT
TYPE typeStationTask :
STRUCT
	//platern data
	PlaternID: UINT;			//identity of the platern
	PlaternIDValid: BOOL;		//indicator

	PlaternNumOps: UINT;		//number of operations the platerns has seen
	PlaternNumOpsValid: BOOL;   //indicator
	
	//reading of data
	DataReadOK: BOOL;			//TRUE if the part data has been read OK
	DataReadNOK: BOOL;			//TRUE if the part data was not read OK

	//part data
	SerialNumber: STRING[32];	//serial number of part
	SerialNumberValid: BOOL;	//indicator
	PartDescription: STRING[32]; //part is?
	PartDescriptionValid:BOOL;		//indicator
	//PartXXXXNumber: STRING[4]; 
	
	//status data
	OKtoBuild: BOOL;			//TRUE if the part is OK to build
	NOKtoBuild: BOOL;			//TRUE if the part is NOK to build
	QuarantinePart: BOOL;		//TRUE if the part is quarantined
	ScrapPart:BOOL;				//TRUE if the part is scrap status
	PartPresent: BOOL;			//TRUE if the part is present in the station (memory or sensor feedback)
	PartComplete:BOOL;			//TRUE if the part is complete


	//process data
	NumberOfRejectAttempts: USINT; 	//number of times the part failed the process
	NumberOfRejectAttemptsValid: BOOL; //indicator
	NumberOfRejectAttemptsFailed: BOOL; //indicator
	LastOperationNumber:UINT;		//last operation number of the previous machine tool
	LastOperationNumberValid: BOOL; //indicator
	
	CycleTimeTarget: REAL :=60.0;	//target cycle time, e.g. 60s
	CycleTimeActual: REAL :=0;		//actual cycle time
	CycleTimePartOver:REAL:=5;		//cycle time is part over, e.g. 5s
	CycleTimeGrossOver:REAL:=120; 	//time for grossly over cycle time
	CycleTimeLast: REAL;			//last part cycle time
	OverCycleTime:BOOL;				//TRUE if over cycle time
	CycleTimeIsGrossOver:BOOL;		//TRUE if cycle time is grossly over
	
	partType:UINT;					//part type
	

	tasks:ARRAY[1..maxNumTasks]  OF typeIndividualTask;	//collection of tasks used in station
END_STRUCT
END_TYPE

// ---- X_DUTs/Tasks/TaskState.TcDUT
{attribute 'qualified_only'}
{attribute 'strict'}
TYPE TaskState :
(
	NoText := 0, 
	NotStarted := 1, 
	Started := 2, 
	Completed := 3,
	Passed := 4,
	Failed := 5,
	Rejected := 6,
	Skipped := 7,
	Bypassed := 8,
	Unknown := 9,
	spare := 10,
	spare1 := 11
		
)USINT;
END_TYPE

// ---- Data Collection/dataGrab.TcGVL
{attribute 'qualified_only'}
VAR_GLOBAL
	//current data being shown
	dataCurrentVisu:structAnalysis;

	data1:structAnalysis;
	data2:structAnalysis;
	data3:structAnalysis;
	
	
END_VAR

// ---- HMI1/Data/gLicenceView.TcGVL
{attribute 'qualified_only'}
VAR_GLOBAL
	
//licences
licenceType:UDINT; //selection from radio button
maxlicenceIndex:UDINT;//max index num
nValidLicences:UDINT;
aValidLicences: ARRAY [1..nMaxLicenses] OF ST_TcOnlineLicenseInfoDataEx;

nPendingLicences:UDINT;
aPendingLicences: ARRAY [1..nMaxLicenses] OF ST_TcOnlineLicenseInfoDataEx;

nDemoLicences:UDINT;
aDemoLicences: ARRAY [1..nMaxLicenses] OF ST_TcOnlineLicenseInfoDataEx;

nOEMLicences:UDINT;
aOEMLicences: ARRAY [1..nMaxLicenses] OF ST_TcOnlineLicenseInfoDataEx;

nFailedLicences:UDINT;
aFailedLicences: ARRAY [1..nMaxLicenses] OF ST_TcOnlineLicenseInfoDataEx;

nInvalidLicences:UDINT;
aInvalidLicences: ARRAY [1..nMaxLicenses] OF ST_TcOnlineLicenseInfoDataEx;

tActiveLicenceSel:UDINT;
tActiveLicenceSelLast:UDINT;
tActiveLicenceArray: ST_TcOnlineLicenseInfoDataEx;
tActiveLicenceList:ARRAY[1..nMaxLicenses] OF STRING(80);
tCallUpdateLicenceList:BOOL; //TRUE to update FB



END_VAR

// ---- HMI1/Data/gModeAlternate.TcGVL
{attribute 'qualified_only'}
VAR_GLOBAL
		//Unit rows and buttons to feedback into program
	gModeRows: typeMotionScreen;
	gModeButtons: typeMotionScreenBtn;
	
END_VAR

// ---- HMI1/Data/TOAST-HMI/gTOASTHMI.TcGVL
{attribute 'qualified_only'}
VAR_GLOBAL
	
	//for reading as
	//dynamic gTOASTHMI = symbols["gTOASTHHMI"];
	gData:structHMIGlobal;
	
END_VAR

// ---- HMI1/Screens/Machine Settings/constCSV.TcGVL
{attribute 'qualified_only'}
VAR_GLOBAL
	DEFAULT_CSV_FIELD_SEP 	: BYTE := 16#2C;(* Comma ASCII code *)
END_VAR

VAR_GLOBAL CONSTANT
	MAX_CSV_ROWS 			: UDINT := 100;
	MAX_CSV_COLUMNS 		: UDINT := 1; //starts from 0
	MAX_CSV_FIELD_LENGTH	: UDINT := 100;
	
	MAX_SETTING_LENGTH		:INT := 100;
	
	str_mc_filelocation		:STRING := 'C:\PLC\machinesettings.csv';
END_VAR

// ---- HMI1/Screens/Machine Settings/MachineSettings.TcGVL
{attribute 'qualified_only'}
VAR_GLOBAL
	
	csvData	: ARRAY[0..constCSV.MAX_CSV_ROWS, 0..constCSV.MAX_CSV_COLUMNS ] OF STRING(constCSV.MAX_CSV_FIELD_LENGTH);
	Setting: ARRAY[0..constcsv.MAX_SETTING_LENGTH] OF typeSettings;
	
	varSelectedColumn:INT;
	varSelectedRow:INT;
	
	varSelectedColumnValid:BOOL;
	varSelectedRowValid:BOOL;
	
	btnRead:BOOL;
	btnWrite:BOOL;
	
	numElementsOfSettings:INT;
	
	numSelectedSetting:INT;
	numSelectedSettingNew:INT;
	btnMoveValue:BOOL;
	
	strStatusFeeback:STRING;
	
	
	
	
	
END_VAR

// ---- HMI1/Screens/Sequences/AutoRowsVisu.TcGVL
{attribute 'qualified_only'}
VAR_GLOBAL
	currentRowNum:UINT;
	currentStepNum:UINT;
END_VAR

// ---- PLC/Safety/Safety.TcGVL
{attribute 'qualified_only'}
VAR_GLOBAL

//mapped from safety CPU EL6910	
gSafetyProgramChecksum	AT %I*	:WORD;		//checksum of user program	
gSafetySerialNumber		AT %I*	:UDINT;		//serial number of safety CPU
gSafetyCPUState			AT %I*	:UINT;		//CPU state as ethercat slave
gSafetyCPUADSadr		AT %I*	:AMSADDR;	//CPU AMSADR

//on request (latch-use) from PLC program to safety program
//this comes from the "Motive Power ON" from the PLC
//otherwise the Safety reset would enable motive power on a _reset_ button
//outputs from PLC (i) program become inputs to safety program (q)
//iEnableSafetyDevices	AT %Q*	:BOOL;
iEnableSafetyDevicesuint	AT %Q*	:UINT;
iEnablePendantSafetyDevicesuint AT %Q*:UINT;

//mapped from safety program
//outputs from PLC (i) program become inputs to safety program (q)
iGroupPort_ErrAck	AT %Q*	:BOOL;
iModuleFault		AT %Q*	:BOOL;
iRunStop			AT %Q*	:BOOL;
iResetFBs			AT %Q*	:BOOL; //seperate reset logic

//outputs from safety program (q) become inputs to PLC program (i) 
qComError			AT %I*	:BOOL;
qCommStartup		AT %I*	:BOOL;
qFBDeactive			AT %I*	:BOOL;
qFBError			AT %I*	:BOOL;
qInRun				AT %I*	:BOOL;
qOtherError			AT %I*	:BOOL;
qOutError			AT %I*	:BOOL;
qRun				AT %I*	:BOOL;

//feedback from program for device evaluation
iEstop1State		AT %I*	:USINT;
iEstop1Diag			AT %I*	:structEstopDiag;

iEstop2State		AT %I*	:USINT;
iEstop2Diag			AT %I*	:structEstopDiag;

iEstop3State		AT %I*	:USINT;
iEstop3Diag			AT %I*	:structEstopDiag;

iAccessGate1State	AT %I*	:USINT;
iAccessGate1Diag	AT %I*	:structEstopDiag;

iAccessGate2State	AT %I*	:USINT;
iAccessGate2Diag	AT %I*	:structEstopDiag;

iEnablingPendantState	AT %I*	:USINT;
iEnablingPendantDiag	AT %I*	:structEstopDiag;


END_VAR

// ---- Version/Global_Version.TcGVL
{attribute 'TcGenerated'}
{attribute 'no-analysis'}
{attribute 'linkalways'}
// This function has been automatically generated from the project information.
VAR_GLOBAL CONSTANT
	{attribute 'const_non_replaced'}
	stLibVersion_Project_Title : ST_LibVersion := (iMajor := 0, iMinor := 0, iBuild := 1, iRevision := 1, nFlags := 0, sVersion := '0.0.1.1');
END_VAR

// ---- HMI1/Data/gHMIButtons.TcGVL
{attribute 'qualified_only'}
VAR_GLOBAL
	//buttons to select a station
	btnSelectStation1: BOOL;
	btnSelectStation2: BOOL;
	btnSelectStation3: BOOL;
	btnSelectStation4: BOOL;
	btnSelectStation5: BOOL;
	btnSelectStation6: BOOL;

	btnSelectAll: BOOL;	//button to select all stations
	btnAllStationsSelected: BOOL;

	//reset button for global use
	btnReset: BOOL;

	//manual screen
	btnAbsMode:BOOL; //TRUE if abs mode, False if sys mode
	btnNextPage: BOOL;
	btnPrevPage: BOOL;
	
	//hide button data for main screen
	btnHides:typeBtnHides;
	
	//hmi buttons
	btnMode:typeBtnPress;
	
	//hmi buttons feedback
	btnFdbk: typeBtnFdbk;
	
	btnPlus1Row:BOOL; //scroll 1 row up
	btnNeg1Row:BOOL; //scroll 1 row down
	clk: INT;
	
	gAnyButtonPressed:BOOL; //TRUE if any button was pressed
	
		//buttons to lock a station
	btnLockStation1: BOOL;
	btnLockStation2: BOOL;
	btnLockStation3: BOOL;
	btnLockStation4: BOOL;
	btnLockStation5: BOOL;
	btnLockStation6: BOOL;
	
	gLockButtons:typeStationLockModes;
	
	gAnyMotionButtonPresed:BOOL; //TRUE if any motion button was pressed
	
	

END_VAR

// ---- HMI1/Data/gHMIDataConst.TcGVL
{attribute 'qualified_only'}
VAR_GLOBAL CONSTANT
	gNumberOfStations: UINT := 6; //number of station in the machine
	gNumberRowsPerPage:UINT := 9; //number of motion rows in the HMI
	gNumberElementsPerRow:UINT := 20;  //number of _things_ in each row, buttons, indicators, etc
	gNumberOfMessagesScreen:UINT:= 100; //number of messages to consider in the alarm screen (number of text lines in alarm view for multiple rows)
END_VAR

// ---- HMI1/Data/gHMIMotionRows.TcGVL
{attribute 'qualified_only'}
VAR_GLOBAL
	//motion rows and buttons to feedback into program
	gMotionRows: typeMotionScreen;
	gMotionRowButtons: typeMotionScreenBtn;
END_VAR

// ---- HMI1/Data/gHMIUnits.TcGVL
{attribute 'qualified_only'}
VAR_GLOBAL
	//Unit rows and buttons to feedback into program
	gUnitRows: typeMotionScreen;
	gUnitButtons: typeMotionScreenBtn;
	gUnitActivePageNumber:UINT; //current page number for units
	gUnitMaxPageNumber:UINT;  //max pages exist for station, e.g. 5
	gUnitActiveStationNumber:UINT; 
	gUnitRowElementOffset: ARRAY[1..gHMIDataConst.gNumberRowsPerPage] OF UINT; //seperate calculation for units

END_VAR

// ---- HMI1/Data/gMsgView.TcGVL
{attribute 'qualified_only'}
VAR_GLOBAL
	
	//nulls do not apply, have to assign to FB
	msgArrynull: ARRAY[1..gHMIDataConst.gNumberOfMessagesScreen] OF typeNewMsg;
	msgArryStylenull: ARRAY[1..gHMIDataConst.gNumberOfMessagesScreen] OF typeNewMsgStyle;
	msgWasChangednull:BOOL;
	
END_VAR

// ---- HMI1/Data/HMIColour.TcGVL
{attribute 'qualified_only'}
VAR_GLOBAL CONSTANT
        colourBlue : DWORD := 16#FF0000FF;
        colourGreen : DWORD := 16#FF00FF00;
        colourYellow : DWORD := 16#FFFFFF00;
        colourGrey : DWORD :=16#88888888;
        colourBlack : DWORD := 16#88000000;
        colourRed: DWORD := 16#FFFF0000;
        colourGreyBackground: DWORD := 16#FFC6C6C6;
		colourPink: DWORD := 16#FFFF00CC;
		colourWhite : DWORD := 16#FFFFFFFF;
END_VAR

// ---- PLC/Machine/GlobalMessages.TcGVL
{attribute 'qualified_only'}
VAR_GLOBAL
	
	//define messages for machine base
	gMsgMc	:typeStationMessage;
	
	//define message for each station
	gMsgS1	:typeStationMessage;
	gMsgS2	:typeStationMessage;
	gMsgS3	:typeStationMessage;
	gMsgS4	:typeStationMessage;
	gMsgS5	:typeStationMessage;
	gMsgS6	:typeStationMessage;
	
	//global memory for retaining status of station
	gMsgMcStat	:typeStationStatus;
	gMsgS1Stat	:typeStationStatus;
	gMsgS2Stat	:typeStationStatus;
	gMsgS3Stat	:typeStationStatus;
	gMsgS4Stat	:typeStationStatus;
	gMsgS5Stat	:typeStationStatus;
	gMsgS6Stat	:typeStationStatus;
	
	//list view of messages in array form
	gListMsgMc	:typeMessageRowsArry;
	gListMsgS1	:typeMessageRowsArry;
	gListMsgS2	:typeMessageRowsArry;
	gListMsgS3	:typeMessageRowsArry;
	gListMsgS4	:typeMessageRowsArry;
	gListMsgS5	:typeMessageRowsArry;
	gListMsgS6	:typeMessageRowsArry;

	gAnyFaultMessage: BOOL; //TRUE if there are any fault messages (any)
	gAnyWarnings: BOOL; //TRUE if there are any warnings (the yellow ones)

	//alarm view of messages in alarmview form
	gMcAlarmView: typeAlarmViewStation;
	gS1AlarmView: typeAlarmViewStation;
	gS2AlarmView: typeAlarmViewStation;
	gS3AlarmView: typeAlarmViewStation;
	gS4AlarmView: typeAlarmViewStation;
	gS5AlarmView: typeAlarmViewStation;
	gS6AlarmView: typeAlarmViewStation;
	
	gHMIAlarmView: typeAlarmViewStation;
	
	//prompt view of messages in alarmview form (not used) test
	gMcPromptView: typeAlarmViewStation;
	gS1PromptView: typeAlarmViewStation;
	gS2PromptView: typeAlarmViewStation;
	gS3PromptView: typeAlarmViewStation;
	gS4PromptView: typeAlarmViewStation;
	gS5PromptView: typeAlarmViewStation;
	gS6PromptView: typeAlarmViewStation;
END_VAR


VAR_GLOBAL CONSTANT
		AllocMsgPerRow:UINT := 10; //number of messages assigned per row
		gNumMessagesPerType:INT := 1000; //number of messages in each type of message
END_VAR

// ---- PLC/Machine/Remote.TcGVL
{attribute 'qualified_only'}
VAR_GLOBAL
	//data to THIS station/machine to be accepted
	ToStation: typeRemote;
	
	//data fed to NEXT or supervisor segment station
	//todo

END_VAR

// ---- PLC/Machine/System.TcGVL
{attribute 'qualified_only'}
VAR_GLOBAL
	
myPlcAppSystemInfo:PlcAppSystemInfo;
myPlcInfoTask1 : PlcTaskSystemInfo;
myPlcInfoTask2 : PlcTaskSystemInfo;
myPlcInfoTask3 : PlcTaskSystemInfo;
myPlcInfoTask4 : PlcTaskSystemInfo;
myPlcInfoTask5 : PlcTaskSystemInfo;
myPlcInfoTask6 : PlcTaskSystemInfo;


ScanTimeReq:REAL; //the programmed task scan time, e.g. 1, 10, 15, 30ms, etc
ScanTimeAct:REAL; //the last scan time, effective current scan time.

ScanTimeRecord:REAL; //the record scan time
ScanTimeRecordScan:LREAL; //the scan number of the record scan time


//EtherCAT masters mapped into all memory
ecMasterData :ARRAY[1..etherCATdiag.maxNumEtherCATmasters] OF typeEtherCATmasters;

thetime: TIMESTRUCT;

oneMilliSecond: BOOL;
hundredMilliSecond:BOOL;
OneSecond: BOOL;
TwoSecond: BOOL;
TenSecond: BOOL;

StartPulse:BOOL;

PulseOneMilliSecond: BOOL;
PulseHundredMilliSecond:BOOL;
PulseOneSecond: BOOL;
PulseTwoSecond: BOOL;
PulseTenSecond: BOOL;

timeDT: DT;

gSetup:typeSetupMachine; //setup data for machine

cpuusageval:UDINT; //CPU usage in percent

symCount: UDINT; //Max. number of available symbols 
sysSize: UDINT; //Max. byte size of symbol information

LatencyMicroSec:UDINT;	//Actual latency in µs 
MaxLatencyMicroSec:UDINT; //Maximum latency in µs

TCRestartReq:BOOL; //restart TC
TCStopReq:BOOL; //stop TC
TCConfigReq:BOOL; //stop TC
NThostname:T_MaxString; //NT hostname
networkadaptors: ARRAY [0..MAX_LOCAL_ADAPTERS] OF ST_IpAdapterInfo;

sysDeviceInfo: Tc2_Utilities.ST_DeviceIdentificationEx;
sysDeviceUpdate:BOOL;

AmsNetIdstr: STRING(23);
AmsNetIdbytes: ARRAY[0..5] OF BYTE;

gHappyBirthday:BOOL;


END_VAR

// ---- HMI1/Data/gHMIData.TcGVL
{attribute 'qualified_only'}
VAR_GLOBAL
	//station selected as BOOL
	gStationSelected: ARRAY[1..gHMIDataConst.gNumberOfStations] OF BOOL;
	
	//hide display elements
	gHideDisplayElements:ARRAY[0..gHMIDataConst.gNumberOfStations] OF BOOL;
	
	//stations enabled
	gStationEnabled: ARRAY[1..gHMIDataConst.gNumberOfStations] OF BOOL;
	
	gRowElementOffset: ARRAY[1..gHMIDataConst.gNumberRowsPerPage] OF UINT;
	
	//number of the active station for message display
	gNumActivePromptTextList:ARRAY[0..gHMIDataConst.gNumberOfStations] OF UINT;
	gNumActiveWarningTextList:ARRAY[0..gHMIDataConst.gNumberOfStations] OF UINT;
	gNumActiveAlarmTextList:ARRAY[0..gHMIDataConst.gNumberOfStations] OF UINT;
	
	//station selected as integer
	gActiveStationNumber:UINT; 
	
	gActivePageNumber:UINT; //current page number
	gMaxPageNumber:UINT;  //max pages exist for station, e.g. 5
	
	gActiveScreen:UINT; //combo of station + page, expressed as integer 0-999999+, reference to the text list
	
	//machine prompt number to display (summation)
	gMachinePromptNumber: UINT;

	//current number of screen on HMI
	gScreenNumber: UINT;

	//hide display elements based on what station is selected
	gHideDisplayElementAlarmView: typeStationEnables;
	gHideDisplayElementWarningView: typeStationEnables;
	gHideDisplayElementPromptView: typeStationEnables;
	
	
	gAlarmViewMsg: typeMessageRowsArry; //connect data to the HMI
	
	//header data
	hmiHeader:typeHMIheader;
	
	//language screen
	gLangRowElementOffset: ARRAY[1..gHMIDataConst.gNumberRowsPerPage] OF UINT; //seperate calculation for languages
	gLangRows: typeMotionScreen;
	gLangButtons: typeMotionScreenBtn;
	gActiveLangPageNumber:UINT; //current page number for units
	gMaxPageNumberLang:UINT;  //max pages exist for station, e.g. 5
	
	gHMIScreenString:STRING;
	
	//title of manual motion screen
	gManualScreenTitle:UINT;
	
	gVisuHasInited:BOOL;
	
	//buttons to lock a station
	gStateLockStation1: USINT;
	gStateLockStation2: USINT;
	gStateLockStation3: USINT;
	gStateLockStation4: USINT;
	gStateLockStation5: USINT;
	gStateLockStation6: USINT;
	
END_VAR

// ---- X_DUTs/Tasks/Tasks.TcGVL
VAR_GLOBAL
END_VAR


VAR_GLOBAL CONSTANT
	maxNumTasks: UINT := 20; //max number of tasks in the station.
END_VAR

// ---- Data Collection/task/taskDataGrab.TcPOU
PROGRAM taskDataGrab
VAR
END_VAR

//call the data grab
prgDataGrab();

END_PROGRAM

// ---- Data Collection/prgDataGrab.TcPOU
PROGRAM prgDataGrab
VAR
	tGrabData: BOOL;
	
	DataIndex: ULINT;
	MaxAxisGrab: ULINT;
	tAxisFull: BOOL;
	
	visuBoxControl1:FB_BoxControl;
	visuBoxControl2:FB_BoxControl;
	visuBoxControl3:FB_BoxControl;
	
	CheckWindow1:FB_Window;
	
END_VAR

actPopulateAxis();


//temp control boxes
//change the button control function on the boxes
visuBoxControl1(iqBoxdata := dataGrab.dataCurrentVisu.box1);
visuBoxControl2(iqBoxdata := dataGrab.dataCurrentVisu.box2);
visuBoxControl3(iqBoxdata := dataGrab.dataCurrentVisu.box3);


CheckWindow1(	dataAxis		:=	dataGrab.dataCurrentVisu.axis,
				i1				:=	datagrab.dataCurrentVisu.box1.i1, //co-ords
				i2				:=	datagrab.dataCurrentVisu.box1.i2, //co-ords
				i3				:=	datagrab.dataCurrentVisu.box1.i3, //co-ords
				i4				:=	datagrab.dataCurrentVisu.box1.i4, //co-ords
				LeftPermSide	:=	datagrab.dataCurrentVisu.box1.leftStatus,
				RightPermSide	:=	datagrab.dataCurrentVisu.box1.rightStatus,
				TopPermSide		:=	datagrab.dataCurrentVisu.box1.topStatus,
				BottomPermSide	:=	datagrab.dataCurrentVisu.box1.bottomStatus
				);

ACTION actPopulateAxis:
MaxAxisGrab := 100;

//populate axis

(*
IF tGrabData THEN

DataIndex := DataIndex + 1;

	//lets grab data
	IF DataIndex < MaxAxisGrab THEN
		dataGrab.axis1.grabTime[dataIndex] := DataIndex;
		dataGrab.axis1.grabData[dataIndex] := 123.456;
		
		
	END_IF
	
	IF DataIndex >= MaxAxisGrab THEN
		tAxisFull := TRUE;
		tGrabData := FALSE;
	END_IF
	

END_IF


*)
END_ACTION

END_PROGRAM

// ---- Data Collection/dynamicBox/FB_BoxControl.TcPOU
FUNCTION_BLOCK FB_BoxControl
VAR_INPUT
	iMaxNumLimit:USINT:=4;
	
END_VAR
VAR_OUTPUT
END_VAR
VAR
END_VAR
VAR_IN_OUT
		iqBoxdata:structBoxData;
END_VAR
VAR // added by the converter: edge detectors and wires of the graphical bodies
    _rt1, _rt2, _rt3, _rt4 : R_TRIG;
    _w1, _w2, _w3, _w4 : BOOL;
END_VAR

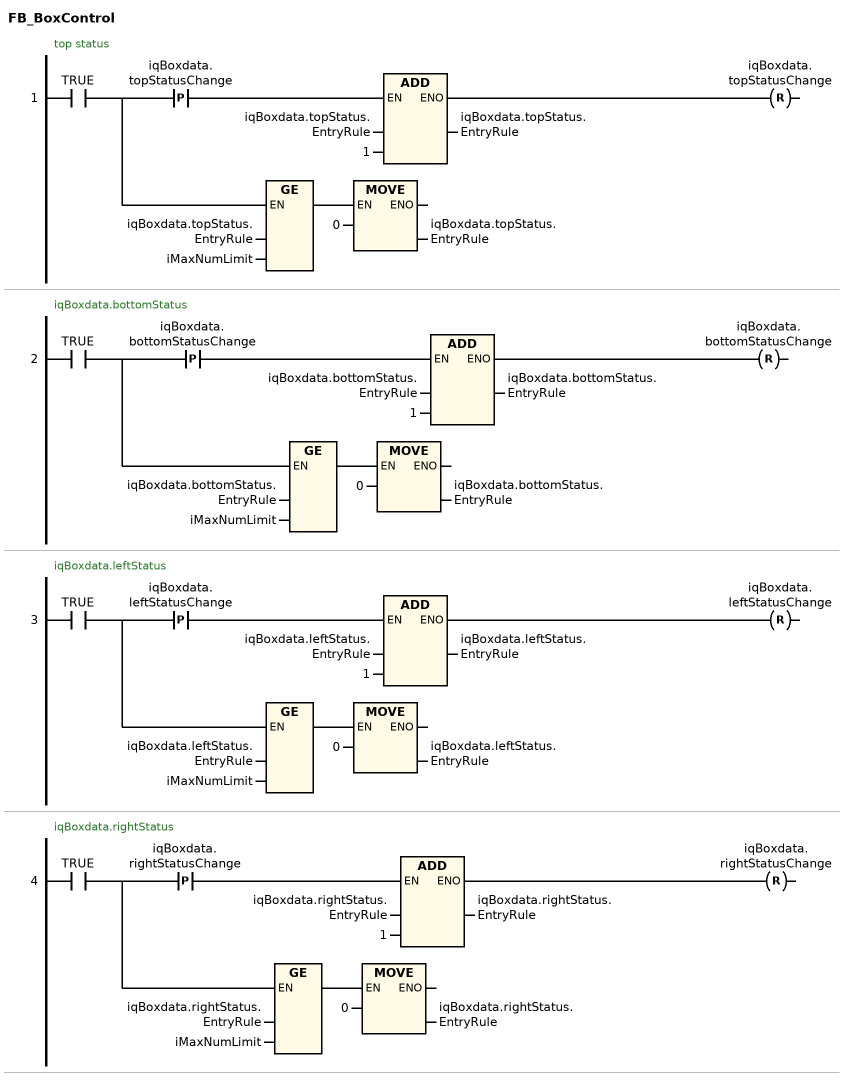
// NETWORK 1
// top status
_rt1(CLK := iqBoxdata.topStatusChange);
_w1 := TRUE AND _rt1.Q;
IF _w1 THEN iqBoxdata.topStatus.EntryRule := iqBoxdata.topStatus.EntryRule + 1; END_IF
iqBoxdata.topStatusChange R= _w1;
IF iqBoxdata.topStatus.EntryRule >= iMaxNumLimit THEN iqBoxdata.topStatus.EntryRule := 0; END_IF

// NETWORK 2
// iqBoxdata.bottomStatus
_rt2(CLK := iqBoxdata.bottomStatusChange);
_w2 := TRUE AND _rt2.Q;
IF _w2 THEN iqBoxdata.bottomStatus.EntryRule := iqBoxdata.bottomStatus.EntryRule + 1; END_IF
iqBoxdata.bottomStatusChange R= _w2;
IF iqBoxdata.bottomStatus.EntryRule >= iMaxNumLimit THEN iqBoxdata.bottomStatus.EntryRule := 0; END_IF

// NETWORK 3
// iqBoxdata.leftStatus
_rt3(CLK := iqBoxdata.leftStatusChange);
_w3 := TRUE AND _rt3.Q;
IF _w3 THEN iqBoxdata.leftStatus.EntryRule := iqBoxdata.leftStatus.EntryRule + 1; END_IF
iqBoxdata.leftStatusChange R= _w3;
IF iqBoxdata.leftStatus.EntryRule >= iMaxNumLimit THEN iqBoxdata.leftStatus.EntryRule := 0; END_IF

// NETWORK 4
// iqBoxdata.rightStatus
_rt4(CLK := iqBoxdata.rightStatusChange);
_w4 := TRUE AND _rt4.Q;
IF _w4 THEN iqBoxdata.rightStatus.EntryRule := iqBoxdata.rightStatus.EntryRule + 1; END_IF
iqBoxdata.rightStatusChange R= _w4;
IF iqBoxdata.rightStatus.EntryRule >= iMaxNumLimit THEN iqBoxdata.rightStatus.EntryRule := 0; END_IF

END_FUNCTION_BLOCK

// ---- Data Collection/dataAnalyse/FB_Window.TcPOU
FUNCTION_BLOCK FB_Window
VAR
    i : DINT; //loop counter
    SampleSpansBoxTime  : BOOL; //check if the data sample was an edge case between lines
    EnteredViaValidSide : BOOL; //TRUE if the line was a valid entry
    HasExitedBox        : BOOL; //TRUE if the line exited the box
    PermissionViolation : BOOL; // Flagged if it passes through an unpermitted line
    ValidEntrySide      : INT;  // 1 = Side A, 3 = Side C, 4 = Side D
    TrappedSuccessfully : BOOL; 
	
	osrStartAnalysis:R_TRIG;
	
END_VAR
VAR_INPUT
	//data to check
	dataAxis: typeDataAxis;

    // Corner Points
    i1 : ST_BoxCorner; // Top-Left
    i2 : ST_BoxCorner; // Bottom-Left
    i3 : ST_BoxCorner; // Bottom-Right
    i4 : ST_BoxCorner; // Top-Right

    // Wall Permissions 
    LeftPermSide : ST_WallPermission; // Left Wall Permissions
    RightPermSide : ST_WallPermission; // Right Wall Permissions
    TopPermSide : ST_WallPermission; // Top Wall Permissions
    BottomPermSide : ST_WallPermission; // Bottom Wall Permissions
	
	iPerformAnalysis:BOOL;
		
END_VAR

VAR_OUTPUT
    qPass : BOOL; // TRUE if data entered legally and followed all rules
    qFail : BOOL; // TRUE if any permission rule was violated or it leaked out
	qErrorCode : E_BoxResultCode; //diag codes
END_VAR

// Reset tracking variables before running the historical loop
EnteredViaValidSide := FALSE;
HasExitedBox        := FALSE;
PermissionViolation := FALSE;
ValidEntrySide      := 0; 
qPass               := FALSE;
qFail               := FALSE;
qErrorCode          := E_BoxResultCode.Success; // Default to Success state

osrStartAnalysis(clk := iPerformAnalysis);

IF osrStartAnalysis.Q THEN


// CRITICAL FIX: Cap dynamic loops safely to actual array limit 
FOR i := 2 TO 20000 DO
    
    SampleSpansBoxTime := (dataAxis.grabTime[i] >= i2.PointXTime) AND (dataAxis.grabTime[i-1] <= i3.PointXTime);

    // =========================================================================
    // PART 1: ENTRY DETECTION & ENUM ENTRY CONFIG CHECKS
    // =========================================================================
    IF NOT EnteredViaValidSide AND NOT PermissionViolation THEN
        
        // 1. SIDE A ENTRY (Left Wall)
        IF (dataAxis.grabTime[i-1] < i2.PointXTime) AND (dataAxis.grabTime[i] >= i2.PointXTime) THEN
            IF (dataAxis.grabData[i] > i2.PointYValue) AND (dataAxis.grabData[i] < i1.PointYValue) THEN
                
                IF LeftPermSide.EntryRule = E_WallEntryRule.MustNotEnter THEN
                    PermissionViolation := TRUE;
                    qErrorCode          := E_BoxResultCode.Err_IllegalEntry_SideA;
                ELSE
                    EnteredViaValidSide := TRUE;
                    ValidEntrySide      := 1; // Mapped to Side A
                END_IF
            END_IF
        END_IF

        // 2. SIDE D ENTRY (Bottom Wall)
        IF (dataAxis.grabTime[i] >= i2.PointXTime) AND (dataAxis.grabTime[i] <= i3.PointXTime) THEN
            IF (dataAxis.grabData[i-1] < i2.PointYValue) AND (dataAxis.grabData[i] >= i2.PointYValue) THEN
                
                IF BottomPermSide.EntryRule = E_WallEntryRule.MustNotEnter THEN
                    PermissionViolation := TRUE;
                    qErrorCode          := E_BoxResultCode.Err_IllegalEntry_SideD;
                ELSE
                    EnteredViaValidSide := TRUE;
                    ValidEntrySide      := 4; // Mapped to Side D
                END_IF
            END_IF
        END_IF
		
        // 3. SIDE C ENTRY (Top Wall)
        IF (dataAxis.grabTime[i] >= i2.PointXTime) AND (dataAxis.grabTime[i] <= i3.PointXTime) THEN
            IF (dataAxis.grabData[i-1] > i1.PointYValue) AND (dataAxis.grabData[i] <= i1.PointYValue) THEN
                
                IF TopPermSide.EntryRule = E_WallEntryRule.MustNotEnter THEN
                    PermissionViolation := TRUE;
                    qErrorCode          := E_BoxResultCode.Err_IllegalEntry_SideC;
                ELSE
                    EnteredViaValidSide := TRUE;
                    ValidEntrySide      := 3; // Mapped to Side C
                END_IF
            END_IF
        END_IF
        
        // Break out instantly if the curve broke in through an illegal wall
        IF PermissionViolation THEN
            EXIT;
        END_IF
    END_IF

    // =========================================================================
    // PART 2: EXIT VIOLATION DETECTION (Evaluates immediately if Entered)
    // =========================================================================
    IF EnteredViaValidSide THEN 
        
        // 1. EXIT VIA SIDE B (Right Wall)
        IF (dataAxis.grabTime[i-1] <= i3.PointXTime) AND (dataAxis.grabTime[i] > i3.PointXTime) THEN
            IF (dataAxis.grabData[i] > i3.PointYValue) AND (dataAxis.grabData[i] < i4.PointYValue) THEN
                HasExitedBox := TRUE;
                IF RightPermSide.IsNotPermittedToExit THEN
                    PermissionViolation := TRUE;
                    qErrorCode          := E_BoxResultCode.Violation_Exited_SideB;
                ELSE
                    qErrorCode          := E_BoxResultCode.Success; // Valid completion code
                END_IF
            END_IF
        END_IF

        // 2. EXIT VIA SIDE A (Left Wall)
        IF (dataAxis.grabTime[i-1] >= i2.PointXTime) AND (dataAxis.grabTime[i] < i2.PointXTime) THEN
            IF (dataAxis.grabData[i] > i2.PointYValue) AND (dataAxis.grabData[i] < i1.PointYValue) THEN
                HasExitedBox := TRUE;
                IF LeftPermSide.IsNotPermittedToExit THEN
                    PermissionViolation := TRUE;
                    qErrorCode          := E_BoxResultCode.Violation_Exited_SideA;
                ELSE
                    qErrorCode          := E_BoxResultCode.Leak_Exited_SideA;
                END_IF
            END_IF
        END_IF

        // 3. EXIT VIA SIDE C (Top Wall)
        IF SampleSpansBoxTime THEN
            IF (dataAxis.grabData[i-1] <= i1.PointYValue) AND (dataAxis.grabData[i] > i1.PointYValue) THEN
                HasExitedBox := TRUE;
                IF TopPermSide.IsNotPermittedToExit THEN
                    PermissionViolation := TRUE;
                    qErrorCode          := E_BoxResultCode.Violation_Exited_SideC;
                ELSE
                    qErrorCode          := E_BoxResultCode.Leak_Exited_SideC;
                END_IF
            END_IF
        END_IF

        // 4. EXIT VIA SIDE D (Bottom Wall)
        IF SampleSpansBoxTime THEN
            IF (dataAxis.grabData[i-1] >= i2.PointYValue) AND (dataAxis.grabData[i] < i2.PointYValue) THEN
                HasExitedBox := TRUE;
                IF BottomPermSide.IsNotPermittedToExit THEN
                    PermissionViolation := TRUE;
                    qErrorCode          := E_BoxResultCode.Violation_Exited_SideD;
                ELSE
                    qErrorCode          := E_BoxResultCode.Leak_Exited_SideD;
                END_IF
            END_IF
        END_IF
        
        // Break loop early if an exit occurred or a specific permission rule was violated
        IF HasExitedBox OR PermissionViolation THEN
            EXIT; 
        END_IF

    END_IF

END_FOR

// =========================================================================
// PART 3: FINAL EVALUATION & MUTUALLY EXCLUSIVE OUTPUTS
// =========================================================================

// Catch the edge case where the loop finished but the signal never even hit a box boundary
	IF NOT EnteredViaValidSide AND NOT PermissionViolation THEN
		qErrorCode := E_BoxResultCode.Err_NeverEnteredBox;
	END_IF
	
	// CRITICAL FIX: Crosscheck "Must Enter" rules across all sides.
	// If any side was marked "Must Enter", but our actual entry side doesn't match it, fail the test.
	IF EnteredViaValidSide AND NOT PermissionViolation THEN
		IF (LeftPermSide.EntryRule = E_WallEntryRule.MustEnter AND ValidEntrySide <> 1) OR
		   (TopPermSide.EntryRule = E_WallEntryRule.MustEnter AND ValidEntrySide <> 3) OR
		   (BottomPermSide.EntryRule = E_WallEntryRule.MustEnter AND ValidEntrySide <> 4) THEN
			
			PermissionViolation := TRUE;
			qErrorCode          := E_BoxResultCode.Err_WrongEntryWall; 
		END_IF
	END_IF

// Evaluate final pass/fail flags
	IF EnteredViaValidSide AND NOT PermissionViolation AND (qErrorCode = E_BoxResultCode.Success) THEN
		qPass      := TRUE;
		qFail      := FALSE;
	ELSE
		qPass      := FALSE;
		qFail      := TRUE;
	END_IF

END_IF

